QRS_NEXT_CUT()
PTP {E1 35817.24,E2 35817.24}
PTP {X 0,Y 759.922,A -85,B 0,C 180,E1 35817.24,E2 35817.24,E3 0,E4 0,E5 0,E6 0}
QRS_SPEED_INIT()
LIN {X 0,Y 759.922,Z 1164.5,A -85,B 0,C 180,E1 35817.24,E2 35817.24,E3 0,E4 0,E5 0,E6 0} C_VEL
LIN {X 0,Y 759.922,Z 407.653,A -85,B 0,C 180,E1 35817.24,E2 35817.24} C_VEL
LIN {X 0,Y 759.922,Z 399.576,A -85,B 0,C 180,E1 35817.24,E2 35817.24} C_VEL
LIN {X 0,Y 759.901,Z 397.576,A -85,B 0,C 180,E1 35817.09,E2 35817.09} C_VEL
LIN {X 0,Y 759.872,Z 397.569,A -85,B 0,C 180,E1 35814.336,E2 35814.336} C_VEL
LIN {X 0,Y 759.909,Z 397.568,A -85,B 0,C 180,E1 35811.602,E2 35811.602} C_VEL
LIN {X 0,Y 759.872,Z 397.574,A -85,B 0,C 180,E1 35808.77,E2 35808.77} C_VEL
LIN {X 0,Y 759.865,Z 397.569,A -85,B 0,C 180,E1 35806.143,E2 35806.143} C_VEL
LIN {X 0,Y 759.911,Z 397.573,A -85,B 0,C 180,E1 35803.317,E2 35803.317} C_VEL
LIN {X 0,Y 759.856,Z 397.573,A -85,B 0,C 180,E1 35800.554,E2 35800.554} C_VEL
LIN {X 0,Y 759.853,Z 397.571,A -85,B 0,C 180,E1 35798.055,E2 35798.055} C_VEL
LIN {X 0,Y 759.916,Z 397.57,A -85,B 0,C 180,E1 35795.348,E2 35795.348} C_VEL
LIN {X 0,Y 759.849,Z 397.574,A -85,B 0,C 180,E1 35792.489,E2 35792.489} C_VEL
LIN {X 0,Y 759.837,Z 397.573,A -85,B 0,C 180,E1 35790.083,E2 35790.083} C_VEL
LIN {X 0,Y 759.879,Z 397.571,A -85,B 0,C 180,E1 35787.508,E2 35787.508} C_VEL
LIN {X 0,Y 759.851,Z 397.576,A -85,B 0,C 180,E1 35784.527,E2 35784.527} C_VEL
LIN {X 0,Y 759.826,Z 397.575,A -85,B 0,C 180,E1 35782.146,E2 35782.146} C_VEL
LIN {X 0,Y 759.824,Z 397.574,A -85,B 0,C 180,E1 35779.848,E2 35779.848} C_VEL
LIN {X 0,Y 759.866,Z 397.572,A -85,B 0,C 180,E1 35777.337,E2 35777.337} C_VEL
LIN {X 0,Y 759.837,Z 397.577,A -85,B 0,C 180,E1 35774.393,E2 35774.393} C_VEL
LIN {X 0,Y 759.811,Z 397.575,A -85,B 0,C 180,E1 35772.054,E2 35772.054} C_VEL
LIN {X 0,Y 759.805,Z 397.577,A -85,B 0,C 180,E1 35769.777,E2 35769.777} C_VEL
LIN {X 0,Y 759.812,Z 397.577,A -85,B 0,C 180,E1 35767.539,E2 35767.539} C_VEL
LIN {X 0,Y 759.907,Z 397.578,A -85,B 0,C 180,E1 35764.808,E2 35764.808} C_VEL
LIN {X 0,Y 759.82,Z 397.573,A -85,B 0,C 180,E1 35762.061,E2 35762.061} C_VEL
LIN {X 0,Y 759.89,Z 397.819,A -85,B 0,C 180,E1 35760.915,E2 35760.915} C_VEL
LIN {X 0,Y 759.919,Z 413.781,A -85,B 0,C 180,E1 35759.761,E2 35759.761} C_VEL
LIN {X 0,Y 759.908,Z 637.992,A -85,B 0,C 180,E1 35757.315,E2 35757.315} C_VEL
LIN {X 0,Y 759.91,Z 802.101,A -85,B 0,C 180,E1 35755.549,E2 35755.549} C_VEL
LIN {X 0,Y 759.898,Z 825.96,A -85,B 0,C 180,E1 35755.172,E2 35755.172} C_VEL
LIN {X 0,Y 759.907,Z 847.797,A -85,B 0,C 180,E1 35754.694,E2 35754.694} C_VEL
LIN {X 0,Y 759.894,Z 868.493,A -85,B 0,C 180,E1 35754.136,E2 35754.136} C_VEL
LIN {X 0,Y 759.918,Z 893.54,A -85,B 0,C 180,E1 35753.303,E2 35753.303} C_VEL
LIN {X 0,Y 759.919,Z 913.093,A -85,B 0,C 180,E1 35752.529,E2 35752.529} C_VEL
LIN {X 0,Y 759.914,Z 935.14,A -85,B 0,C 180,E1 35751.523,E2 35751.523} C_VEL
LIN {X 0,Y 759.917,Z 955.453,A -85,B 0,C 180,E1 35750.439,E2 35750.439} C_VEL
LIN {X 0,Y 759.91,Z 975.283,A -85,B 0,C 180,E1 35749.245,E2 35749.245} C_VEL
LIN {X 0,Y 759.904,Z 994.198,A -85,B 0,C 180,E1 35747.933,E2 35747.933} C_VEL
LIN {X 0,Y 759.914,Z 1012.37,A -85,B 0,C 180,E1 35746.512,E2 35746.512} C_VEL
LIN {X 0,Y 759.91,Z 1028.199,A -85,B 0,C 180,E1 35745.102,E2 35745.102} C_VEL
LIN {X 0,Y 759.917,Z 1044.372,A -85,B 0,C 180,E1 35743.468,E2 35743.468} C_VEL
LIN {X 0,Y 759.904,Z 1057.076,A -85,B 0,C 180,E1 35741.999,E2 35741.999} C_VEL
LIN {X 0,Y 759.918,Z 1069.916,A -85,B 0,C 180,E1 35740.308,E2 35740.308} C_VEL
LIN {X 0,Y 759.893,Z 1080.292,A -85,B 0,C 180,E1 35738.704,E2 35738.704} C_VEL
LIN {X 0,Y 759.899,Z 1089.216,A -85,B 0,C 180,E1 35737.105,E2 35737.105} C_VEL
LIN {X 0,Y 759.897,Z 1097.567,A -85,B 0,C 180,E1 35735.285,E2 35735.285} C_VEL
LIN {X 0,Y 759.897,Z 1103.433,A -85,B 0,C 180,E1 35733.697,E2 35733.697} C_VEL
LIN {X 0,Y 759.914,Z 1108.651,A -85,B 0,C 180,E1 35731.885,E2 35731.885} C_VEL
LIN {X 0,Y 759.917,Z 1112.079,A -85,B 0,C 180,E1 35730.075,E2 35730.075} C_VEL
LIN {X 0,Y 759.889,Z 1113.939,A -85,B 0,C 180,E1 35728.417,E2 35728.417} C_VEL
LIN {X 0,Y 759.889,Z 1114.381,A -85,B 0,C 180,E1 35726.53,E2 35726.53} C_VEL
LIN {X 0,Y 759.892,Z 1113.442,A -85,B 0,C 180,E1 35724.932,E2 35724.932} C_VEL
LIN {X 0,Y 759.883,Z 1110.795,A -85,B 0,C 180,E1 35723.047,E2 35723.047} C_VEL
LIN {X 0,Y 759.909,Z 1106.908,A -85,B 0,C 180,E1 35721.373,E2 35721.373} C_VEL
LIN {X 0,Y 759.912,Z 1101.686,A -85,B 0,C 180,E1 35719.691,E2 35719.691} C_VEL
LIN {X 0,Y 759.905,Z 1094.199,A -85,B 0,C 180,E1 35717.847,E2 35717.847} C_VEL
LIN {X 0,Y 759.897,Z 1086.525,A -85,B 0,C 180,E1 35716.299,E2 35716.299} C_VEL
LIN {X 0,Y 759.904,Z 1076.531,A -85,B 0,C 180,E1 35714.586,E2 35714.586} C_VEL
LIN {X 0,Y 759.889,Z 1065.053,A -85,B 0,C 180,E1 35712.936,E2 35712.936} C_VEL
LIN {X 0,Y 759.913,Z 1052.308,A -85,B 0,C 180,E1 35711.33,E2 35711.33} C_VEL
LIN {X 0,Y 759.904,Z 1037.754,A -85,B 0,C 180,E1 35709.748,E2 35709.748} C_VEL
LIN {X 0,Y 759.9,Z 1021.891,A -85,B 0,C 180,E1 35708.219,E2 35708.219} C_VEL
LIN {X 0,Y 759.904,Z 1004.859,A -85,B 0,C 180,E1 35706.791,E2 35706.791} C_VEL
LIN {X 0,Y 759.918,Z 986.667,A -85,B 0,C 180,E1 35705.431,E2 35705.431} C_VEL
LIN {X 0,Y 759.913,Z 968.159,A -85,B 0,C 180,E1 35704.223,E2 35704.223} C_VEL
LIN {X 0,Y 759.916,Z 947.899,A -85,B 0,C 180,E1 35703.045,E2 35703.045} C_VEL
LIN {X 0,Y 759.916,Z 926.843,A -85,B 0,C 180,E1 35701.994,E2 35701.994} C_VEL
LIN {X 0,Y 759.917,Z 907.016,A -85,B 0,C 180,E1 35701.125,E2 35701.125} C_VEL
LIN {X 0,Y 759.905,Z 883.717,A -85,B 0,C 180,E1 35700.26,E2 35700.26} C_VEL
LIN {X 0,Y 759.899,Z 865.074,A -85,B 0,C 180,E1 35699.676,E2 35699.676} C_VEL
LIN {X 0,Y 759.905,Z 844.11,A -85,B 0,C 180,E1 35699.125,E2 35699.125} C_VEL
LIN {X 0,Y 759.903,Z 819.274,A -85,B 0,C 180,E1 35698.621,E2 35698.621} C_VEL
LIN {X 0,Y 759.908,Z 798.856,A -85,B 0,C 180,E1 35698.32,E2 35698.32} C_VEL
LIN {X 0,Y 759.909,Z 526.746,A -85,B 0,C 180,E1 35695.394,E2 35695.394} C_VEL
LIN {X 0,Y 759.919,Z 413.481,A -85,B 0,C 180,E1 35694.138,E2 35694.138} C_VEL
LIN {X 0,Y 759.888,Z 397.79,A -85,B 0,C 180,E1 35692.99,E2 35692.99} C_VEL
LIN {X 0,Y 759.814,Z 397.578,A -85,B 0,C 180,E1 35690.437,E2 35690.437} C_VEL
LIN {X 0,Y 759.804,Z 397.578,A -85,B 0,C 180,E1 35688.146,E2 35688.146} C_VEL
LIN {X 0,Y 759.81,Z 397.577,A -85,B 0,C 180,E1 35685.881,E2 35685.881} C_VEL
LIN {X 0,Y 759.854,Z 397.577,A -85,B 0,C 180,E1 35683.416,E2 35683.416} C_VEL
LIN {X 0,Y 759.844,Z 397.575,A -85,B 0,C 180,E1 35680.447,E2 35680.447} C_VEL
LIN {X 0,Y 759.824,Z 397.575,A -85,B 0,C 180,E1 35678.099,E2 35678.099} C_VEL
LIN {X 0,Y 759.824,Z 397.573,A -85,B 0,C 180,E1 35675.843,E2 35675.843} C_VEL
LIN {X 0,Y 759.857,Z 397.576,A -85,B 0,C 180,E1 35673.37,E2 35673.37} C_VEL
LIN {X 0,Y 759.862,Z 397.57,A -85,B 0,C 180,E1 35670.319,E2 35670.319} C_VEL
LIN {X 0,Y 759.836,Z 397.573,A -85,B 0,C 180,E1 35667.833,E2 35667.833} C_VEL
LIN {X 0,Y 759.853,Z 397.575,A -85,B 0,C 180,E1 35665.403,E2 35665.403} C_VEL
LIN {X 0,Y 759.919,Z 397.568,A -85,B 0,C 180,E1 35662.513,E2 35662.513} C_VEL
LIN {X 0,Y 759.85,Z 397.571,A -85,B 0,C 180,E1 35659.801,E2 35659.801} C_VEL
LIN {X 0,Y 759.87,Z 397.575,A -85,B 0,C 180,E1 35657.222,E2 35657.222} C_VEL
LIN {X 0,Y 759.906,Z 397.567,A -85,B 0,C 180,E1 35654.244,E2 35654.244} C_VEL
LIN {X 0,Y 759.858,Z 397.571,A -85,B 0,C 180,E1 35651.538,E2 35651.538} C_VEL
LIN {X 0,Y 759.917,Z 397.577,A -85,B 0,C 180,E1 35648.78,E2 35648.78} C_VEL
LIN {X 0,Y 759.881,Z 397.567,A -85,B 0,C 180,E1 35645.815,E2 35645.815} C_VEL
LIN {X 0,Y 759.887,Z 397.575,A -85,B 0,C 180,E1 35643.017,E2 35643.017} C_VEL
LIN {X 0,Y 759.92,Z 397.564,A -85,B 0,C 180,E1 35640,E2 35640} C_VEL
LIN {X 0,Y 759.876,Z 397.571,A -85,B 0,C 180,E1 35637.209,E2 35637.209} C_VEL
LIN {X 0,Y 759.905,Z 397.574,A -85,B 0,C 180,E1 35634.488,E2 35634.488} C_VEL
LIN {X 0,Y 759.896,Z 397.565,A -85,B 0,C 180,E1 35631.601,E2 35631.601} C_VEL
LIN {X 0,Y 759.911,Z 397.577,A -85,B 0,C 180,E1 35628.694,E2 35628.694} C_VEL
LIN {X 0,Y 759.918,Z 397.563,A -85,B 0,C 180,E1 35625.678,E2 35625.678} C_VEL
LIN {X 0,Y 759.914,Z 397.577,A -85,B 0,C 180,E1 35622.621,E2 35622.621} C_VEL
LIN {X 0,Y 759.911,Z 397.564,A -85,B 0,C 180,E1 35619.593,E2 35619.593} C_VEL
LIN {X 0,Y 759.914,Z 397.577,A -85,B 0,C 180,E1 35616.586,E2 35616.586} C_VEL
LIN {X 0,Y 759.895,Z 397.565,A -85,B 0,C 180,E1 35613.648,E2 35613.648} C_VEL
LIN {X 0,Y 759.902,Z 397.574,A -85,B 0,C 180,E1 35610.738,E2 35610.738} C_VEL
LIN {X 0,Y 759.877,Z 397.571,A -85,B 0,C 180,E1 35607.932,E2 35607.932} C_VEL
LIN {X 0,Y 759.912,Z 397.565,A -85,B 0,C 180,E1 35605.176,E2 35605.176} C_VEL
LIN {X 0,Y 759.896,Z 397.575,A -85,B 0,C 180,E1 35602.262,E2 35602.262} C_VEL
LIN {X 0,Y 759.879,Z 397.568,A -85,B 0,C 180,E1 35599.456,E2 35599.456} C_VEL
LIN {X 0,Y 759.91,Z 397.573,A -85,B 0,C 180,E1 35596.579,E2 35596.579} C_VEL
LIN {X 0,Y 759.863,Z 397.573,A -85,B 0,C 180,E1 35593.801,E2 35593.801} C_VEL
LIN {X 0,Y 759.896,Z 397.567,A -85,B 0,C 180,E1 35591.064,E2 35591.064} C_VEL
LIN {X 0,Y 759.886,Z 397.575,A -85,B 0,C 180,E1 35588.105,E2 35588.105} C_VEL
LIN {X 0,Y 759.913,Z 397.781,A -85,B 0,C 180,E1 35586.49,E2 35586.49} C_VEL
LIN {X 0,Y 759.908,Z 427.098,A -85,B 0,C 180,E1 35584.501,E2 35584.501} C_VEL
LIN {X 0,Y 759.907,Z 453.003,A -85,B 0,C 180,E1 35582.815,E2 35582.815} C_VEL
LIN {X 0,Y 759.893,Z 698.451,A -85,B 0,C 180,E1 35580.142,E2 35580.142} C_VEL
LIN {X 0,Y 759.92,Z 841.979,A -85,B 0,C 180,E1 35578.595,E2 35578.595} C_VEL
LIN {X 0,Y 759.894,Z 866.292,A -85,B 0,C 180,E1 35578.211,E2 35578.211} C_VEL
LIN {X 0,Y 759.9,Z 887.681,A -85,B 0,C 180,E1 35577.742,E2 35577.742} C_VEL
LIN {X 0,Y 759.897,Z 907.094,A -85,B 0,C 180,E1 35577.221,E2 35577.221} C_VEL
LIN {X 0,Y 759.919,Z 929.734,A -85,B 0,C 180,E1 35576.491,E2 35576.491} C_VEL
LIN {X 0,Y 759.916,Z 951.248,A -85,B 0,C 180,E1 35575.652,E2 35575.652} C_VEL
LIN {X 0,Y 759.913,Z 970.659,A -85,B 0,C 180,E1 35574.783,E2 35574.783} C_VEL
LIN {X 0,Y 759.91,Z 993.058,A -85,B 0,C 180,E1 35573.62,E2 35573.62} C_VEL
LIN {X 0,Y 759.92,Z 1011.704,A -85,B 0,C 180,E1 35572.513,E2 35572.513} C_VEL
LIN {X 0,Y 759.906,Z 1031.522,A -85,B 0,C 180,E1 35571.173,E2 35571.173} C_VEL
LIN {X 0,Y 759.916,Z 1048.884,A -85,B 0,C 180,E1 35569.845,E2 35569.845} C_VEL
LIN {X 0,Y 759.917,Z 1065.39,A -85,B 0,C 180,E1 35568.409,E2 35568.409} C_VEL
LIN {X 0,Y 759.895,Z 1079.946,A -85,B 0,C 180,E1 35566.985,E2 35566.985} C_VEL
LIN {X 0,Y 759.899,Z 1094.876,A -85,B 0,C 180,E1 35565.312,E2 35565.312} C_VEL
LIN {X 0,Y 759.905,Z 1106.572,A -85,B 0,C 180,E1 35563.815,E2 35563.815} C_VEL
LIN {X 0,Y 759.9,Z 1118.785,A -85,B 0,C 180,E1 35561.999,E2 35561.999} C_VEL
LIN {X 0,Y 759.907,Z 1127.555,A -85,B 0,C 180,E1 35560.462,E2 35560.462} C_VEL
LIN {X 0,Y 759.888,Z 1136.073,A -85,B 0,C 180,E1 35558.704,E2 35558.704} C_VEL
LIN {X 0,Y 759.918,Z 1142.726,A -85,B 0,C 180,E1 35556.953,E2 35556.953} C_VEL
LIN {X 0,Y 759.883,Z 1147.51,A -85,B 0,C 180,E1 35555.361,E2 35555.361} C_VEL
LIN {X 0,Y 759.919,Z 1151.559,A -85,B 0,C 180,E1 35553.47,E2 35553.47} C_VEL
LIN {X 0,Y 759.902,Z 1153.63,A -85,B 0,C 180,E1 35551.81,E2 35551.81} C_VEL
LIN {X 0,Y 759.92,Z 1154.5,A -85,B 0,C 180,E1 35550,E2 35550} C_VEL
LIN {X 0,Y 759.902,Z 1153.63,A -85,B 0,C 180,E1 35548.19,E2 35548.19} C_VEL
LIN {X 0,Y 759.919,Z 1151.559,A -85,B 0,C 180,E1 35546.53,E2 35546.53} C_VEL
LIN {X 0,Y 759.883,Z 1147.51,A -85,B 0,C 180,E1 35544.639,E2 35544.639} C_VEL
LIN {X 0,Y 759.918,Z 1142.726,A -85,B 0,C 180,E1 35543.047,E2 35543.047} C_VEL
LIN {X 0,Y 759.889,Z 1135.729,A -85,B 0,C 180,E1 35541.22,E2 35541.22} C_VEL
LIN {X 0,Y 759.907,Z 1127.555,A -85,B 0,C 180,E1 35539.538,E2 35539.538} C_VEL
LIN {X 0,Y 759.9,Z 1118.785,A -85,B 0,C 180,E1 35538.001,E2 35538.001} C_VEL
LIN {X 0,Y 759.904,Z 1106.265,A -85,B 0,C 180,E1 35536.144,E2 35536.144} C_VEL
LIN {X 0,Y 759.9,Z 1094.679,A -85,B 0,C 180,E1 35534.664,E2 35534.664} C_VEL
LIN {X 0,Y 759.896,Z 1079.169,A -85,B 0,C 180,E1 35532.937,E2 35532.937} C_VEL
LIN {X 0,Y 759.914,Z 1064.539,A -85,B 0,C 180,E1 35531.512,E2 35531.512} C_VEL
LIN {X 0,Y 759.913,Z 1046.484,A -85,B 0,C 180,E1 35529.965,E2 35529.965} C_VEL
LIN {X 0,Y 759.91,Z 1029.578,A -85,B 0,C 180,E1 35528.684,E2 35528.684} C_VEL
LIN {X 0,Y 759.918,Z 1009.719,A -85,B 0,C 180,E1 35527.364,E2 35527.364} C_VEL
LIN {X 0,Y 759.91,Z 990.877,A -85,B 0,C 180,E1 35526.257,E2 35526.257} C_VEL
LIN {X 0,Y 759.913,Z 969.006,A -85,B 0,C 180,E1 35525.14,E2 35525.14} C_VEL
LIN {X 0,Y 759.917,Z 950.063,A -85,B 0,C 180,E1 35524.299,E2 35524.299} C_VEL
LIN {X 0,Y 759.915,Z 927.316,A -85,B 0,C 180,E1 35523.425,E2 35523.425} C_VEL
LIN {X 0,Y 759.899,Z 906.002,A -85,B 0,C 180,E1 35522.748,E2 35522.748} C_VEL
LIN {X 0,Y 759.898,Z 886.063,A -85,B 0,C 180,E1 35522.218,E2 35522.218} C_VEL
LIN {X 0,Y 759.898,Z 861.401,A -85,B 0,C 180,E1 35521.701,E2 35521.701} C_VEL
LIN {X 0,Y 759.92,Z 840.267,A -85,B 0,C 180,E1 35521.383,E2 35521.383} C_VEL
LIN {X 0,Y 759.85,Z 582.634,A -85,B 0,C 180,E1 35518.608,E2 35518.608} C_VEL
LIN {X 0,Y 759.905,Z 452.847,A -85,B 0,C 180,E1 35517.179,E2 35517.179} C_VEL
LIN {X 0,Y 759.916,Z 411.18,A -85,B 0,C 180,E1 35514.438,E2 35514.438} C_VEL
LIN {X 0,Y 759.913,Z 397.769,A -85,B 0,C 180,E1 35513.506,E2 35513.506} C_VEL
LIN {X 0,Y 759.864,Z 397.57,A -85,B 0,C 180,E1 35510.691,E2 35510.691} C_VEL
LIN {X 0,Y 759.871,Z 397.575,A -85,B 0,C 180,E1 35508.028,E2 35508.028} C_VEL
LIN {X 0,Y 759.912,Z 397.568,A -85,B 0,C 180,E1 35505.149,E2 35505.149} C_VEL
LIN {X 0,Y 759.866,Z 397.57,A -85,B 0,C 180,E1 35502.356,E2 35502.356} C_VEL
LIN {X 0,Y 759.915,Z 397.578,A -85,B 0,C 180,E1 35499.551,E2 35499.551} C_VEL
LIN {X 0,Y 759.892,Z 397.566,A -85,B 0,C 180,E1 35496.589,E2 35496.589} C_VEL
LIN {X 0,Y 759.894,Z 397.575,A -85,B 0,C 180,E1 35493.73,E2 35493.73} C_VEL
LIN {X 0,Y 759.909,Z 397.565,A -85,B 0,C 180,E1 35490.771,E2 35490.771} C_VEL
LIN {X 0,Y 759.881,Z 397.57,A -85,B 0,C 180,E1 35488.001,E2 35488.001} C_VEL
LIN {X 0,Y 759.902,Z 397.573,A -85,B 0,C 180,E1 35485.235,E2 35485.235} C_VEL
LIN {X 0,Y 759.9,Z 397.565,A -85,B 0,C 180,E1 35482.328,E2 35482.328} C_VEL
LIN {X 0,Y 759.911,Z 397.577,A -85,B 0,C 180,E1 35479.364,E2 35479.364} C_VEL
LIN {X 0,Y 759.915,Z 397.563,A -85,B 0,C 180,E1 35476.355,E2 35476.355} C_VEL
LIN {X 0,Y 759.915,Z 397.577,A -85,B 0,C 180,E1 35473.313,E2 35473.313} C_VEL
LIN {X 0,Y 759.91,Z 397.564,A -85,B 0,C 180,E1 35470.309,E2 35470.309} C_VEL
LIN {X 0,Y 759.913,Z 397.577,A -85,B 0,C 180,E1 35467.257,E2 35467.257} C_VEL
LIN {X 0,Y 759.89,Z 397.566,A -85,B 0,C 180,E1 35464.377,E2 35464.377} C_VEL
LIN {X 0,Y 759.904,Z 397.573,A -85,B 0,C 180,E1 35461.508,E2 35461.508} C_VEL
LIN {X 0,Y 759.876,Z 397.572,A -85,B 0,C 180,E1 35458.794,E2 35458.794} C_VEL
LIN {X 0,Y 759.901,Z 397.576,A -85,B 0,C 180,E1 35457.09,E2 35457.09} C_VEL
LIN {X 0,Y 758.866,Z 397.696,A -85,B 0,C 180,E1 35456.509,E2 35456.509} C_VEL
LIN {X 0,Y 752.45,Z 398.503,A -85,B 0,C 180,E1 35454.882,E2 35454.882} C_VEL
LIN {X 0,Y 751.929,Z 398.559,A -85,B 0,C 180,E1 35454.46,E2 35454.46} C_VEL
LIN {X 0,Y 751.974,Z 398.554,A -85,B 0,C 180,E1 35451.743,E2 35451.743} C_VEL
LIN {X 0,Y 751.937,Z 398.563,A -85,B 0,C 180,E1 35448.805,E2 35448.805} C_VEL
LIN {X 0,Y 751.929,Z 398.557,A -85,B 0,C 180,E1 35446.105,E2 35446.105} C_VEL
LIN {X 0,Y 751.975,Z 398.564,A -85,B 0,C 180,E1 35443.212,E2 35443.212} C_VEL
LIN {X 0,Y 751.915,Z 398.562,A -85,B 0,C 180,E1 35440.502,E2 35440.502} C_VEL
LIN {X 0,Y 751.922,Z 398.559,A -85,B 0,C 180,E1 35437.951,E2 35437.951} C_VEL
LIN {X 0,Y 751.977,Z 398.564,A -85,B 0,C 180,E1 35435.07,E2 35435.07} C_VEL
LIN {X 0,Y 751.903,Z 398.562,A -85,B 0,C 180,E1 35432.333,E2 35432.333} C_VEL
LIN {X 0,Y 751.905,Z 398.561,A -85,B 0,C 180,E1 35429.911,E2 35429.911} C_VEL
LIN {X 0,Y 751.979,Z 398.562,A -85,B 0,C 180,E1 35427.145,E2 35427.145} C_VEL
LIN {X 0,Y 751.897,Z 398.564,A -85,B 0,C 180,E1 35424.344,E2 35424.344} C_VEL
LIN {X 0,Y 751.886,Z 398.564,A -85,B 0,C 180,E1 35421.996,E2 35421.996} C_VEL
LIN {X 0,Y 751.899,Z 398.563,A -85,B 0,C 180,E1 35419.637,E2 35419.637} C_VEL
LIN {X 0,Y 751.953,Z 398.566,A -85,B 0,C 180,E1 35416.777,E2 35416.777} C_VEL
LIN {X 0,Y 751.881,Z 398.566,A -85,B 0,C 180,E1 35414.175,E2 35414.175} C_VEL
LIN {X 0,Y 751.87,Z 398.561,A -85,B 0,C 180,E1 35411.864,E2 35411.864} C_VEL
LIN {X 0,Y 751.878,Z 398.567,A -85,B 0,C 180,E1 35409.527,E2 35409.527} C_VEL
LIN {X 0,Y 751.953,Z 398.568,A -85,B 0,C 180,E1 35406.695,E2 35406.695} C_VEL
LIN {X 0,Y 751.876,Z 398.568,A -85,B 0,C 180,E1 35404.047,E2 35404.047} C_VEL
LIN {X 0,Y 751.871,Z 398.558,A -85,B 0,C 180,E1 35401.811,E2 35401.811} C_VEL
LIN {X 0,Y 751.955,Z 398.922,A -85,B 0,C 180,E1 35401.234,E2 35401.234} C_VEL
LIN {X 0,Y 752.71,Z 402.275,A -85,B 0,C 180,E1 35400.937,E2 35400.937} C_VEL
LIN {X 0,Y 752.755,Z 413.762,A -85,B 0,C 180,E1 35400.114,E2 35400.114} C_VEL
LIN {X 0,Y 753.183,Z 417.042,A -85,B 0,C 180,E1 35400.046,E2 35400.046} C_VEL
LIN {X 0,Y 752.967,Z 667.075,A -85,B 0,C 180,E1 35397.31,E2 35397.31} C_VEL
LIN {X 0,Y 752.873,Z 802.384,A -85,B 0,C 180,E1 35395.838,E2 35395.838} C_VEL
LIN {X 0,Y 752.802,Z 827.22,A -85,B 0,C 180,E1 35395.436,E2 35395.436} C_VEL
LIN {X 0,Y 752.759,Z 848.615,A -85,B 0,C 180,E1 35394.96,E2 35394.96} C_VEL
LIN {X 0,Y 752.686,Z 870.446,A -85,B 0,C 180,E1 35394.361,E2 35394.361} C_VEL
LIN {X 0,Y 752.612,Z 894.301,A -85,B 0,C 180,E1 35393.55,E2 35393.55} C_VEL
LIN {X 0,Y 752.545,Z 914.316,A -85,B 0,C 180,E1 35392.746,E2 35392.746} C_VEL
LIN {X 0,Y 752.433,Z 937.119,A -85,B 0,C 180,E1 35391.68,E2 35391.68} C_VEL
LIN {X 0,Y 752.364,Z 955.766,A -85,B 0,C 180,E1 35390.671,E2 35390.671} C_VEL
LIN {X 0,Y 752.265,Z 976.401,A -85,B 0,C 180,E1 35389.408,E2 35389.408} C_VEL
LIN {X 0,Y 752.195,Z 994.827,A -85,B 0,C 180,E1 35388.112,E2 35388.112} C_VEL
LIN {X 0,Y 752.126,Z 1013.684,A -85,B 0,C 180,E1 35386.608,E2 35386.608} C_VEL
LIN {X 0,Y 752.076,Z 1029.403,A -85,B 0,C 180,E1 35385.184,E2 35385.184} C_VEL
LIN {X 0,Y 752.026,Z 1045.376,A -85,B 0,C 180,E1 35383.533,E2 35383.533} C_VEL
LIN {X 0,Y 751.983,Z 1057.987,A -85,B 0,C 180,E1 35382.05,E2 35382.05} C_VEL
LIN {X 0,Y 751.962,Z 1071.168,A -85,B 0,C 180,E1 35380.264,E2 35380.264} C_VEL
LIN {X 0,Y 751.923,Z 1080.95,A -85,B 0,C 180,E1 35378.719,E2 35378.719} C_VEL
LIN {X 0,Y 751.904,Z 1090.572,A -85,B 0,C 180,E1 35376.951,E2 35376.951} C_VEL
LIN {X 0,Y 751.912,Z 1098.3,A -85,B 0,C 180,E1 35375.188,E2 35375.188} C_VEL
LIN {X 0,Y 751.892,Z 1104.048,A -85,B 0,C 180,E1 35373.583,E2 35373.583} C_VEL
LIN {X 0,Y 751.914,Z 1109.351,A -85,B 0,C 180,E1 35371.6,E2 35371.6} C_VEL
LIN {X 0,Y 751.914,Z 1112.352,A -85,B 0,C 180,E1 35369.924,E2 35369.924} C_VEL
LIN {X 0,Y 751.917,Z 1114.196,A -85,B 0,C 180,E1 35368.019,E2 35368.019} C_VEL
LIN {X 0,Y 751.889,Z 1114.327,A -85,B 0,C 180,E1 35366.34,E2 35366.34} C_VEL
LIN {X 0,Y 751.911,Z 1113.154,A -85,B 0,C 180,E1 35364.582,E2 35364.582} C_VEL
LIN {X 0,Y 751.884,Z 1110.249,A -85,B 0,C 180,E1 35362.742,E2 35362.742} C_VEL
LIN {X 0,Y 751.916,Z 1106.613,A -85,B 0,C 180,E1 35361.203,E2 35361.203} C_VEL
LIN {X 0,Y 751.902,Z 1100.739,A -85,B 0,C 180,E1 35359.339,E2 35359.339} C_VEL
LIN {X 0,Y 751.915,Z 1093.328,A -85,B 0,C 180,E1 35357.559,E2 35357.559} C_VEL
LIN {X 0,Y 751.921,Z 1085.11,A -85,B 0,C 180,E1 35355.916,E2 35355.916} C_VEL
LIN {X 0,Y 751.944,Z 1074.199,A -85,B 0,C 180,E1 35354.102,E2 35354.102} C_VEL
LIN {X 0,Y 751.96,Z 1063.623,A -85,B 0,C 180,E1 35352.591,E2 35352.591} C_VEL
LIN {X 0,Y 751.998,Z 1049.393,A -85,B 0,C 180,E1 35350.827,E2 35350.827} C_VEL
LIN {X 0,Y 752.048,Z 1035.881,A -85,B 0,C 180,E1 35349.37,E2 35349.37} C_VEL
LIN {X 0,Y 752.119,Z 1019.142,A -85,B 0,C 180,E1 35347.776,E2 35347.776} C_VEL
LIN {X 0,Y 752.158,Z 1002.853,A -85,B 0,C 180,E1 35346.413,E2 35346.413} C_VEL
LIN {X 0,Y 752.247,Z 983.216,A -85,B 0,C 180,E1 35344.966,E2 35344.966} C_VEL
LIN {X 0,Y 752.312,Z 965.042,A -85,B 0,C 180,E1 35343.785,E2 35343.785} C_VEL
LIN {X 0,Y 752.417,Z 943.077,A -85,B 0,C 180,E1 35342.54,E2 35342.54} C_VEL
LIN {X 0,Y 752.49,Z 923.974,A -85,B 0,C 180,E1 35341.595,E2 35341.595} C_VEL
LIN {X 0,Y 752.6,Z 900.73,A -85,B 0,C 180,E1 35340.604,E2 35340.604} C_VEL
LIN {X 0,Y 752.644,Z 879.969,A -85,B 0,C 180,E1 35339.856,E2 35339.856} C_VEL
LIN {X 0,Y 752.741,Z 857.575,A -85,B 0,C 180,E1 35339.176,E2 35339.176} C_VEL
LIN {X 0,Y 752.792,Z 834.253,A -85,B 0,C 180,E1 35338.62,E2 35338.62} C_VEL
LIN {X 0,Y 752.846,Z 814.363,A -85,B 0,C 180,E1 35338.249,E2 35338.249} C_VEL
LIN {X 0,Y 752.88,Z 789.412,A -85,B 0,C 180,E1 35337.912,E2 35337.912} C_VEL
LIN {X 0,Y 753.078,Z 533.824,A -85,B 0,C 180,E1 35335.152,E2 35335.152} C_VEL
LIN {X 0,Y 752.996,Z 414.882,A -85,B 0,C 180,E1 35333.83,E2 35333.83} C_VEL
LIN {X 0,Y 752.683,Z 412.464,A -85,B 0,C 180,E1 35333.718,E2 35333.718} C_VEL
LIN {X 0,Y 752.569,Z 400.863,A -85,B 0,C 180,E1 35332.862,E2 35332.862} C_VEL
LIN {X 0,Y 751.903,Z 398.647,A -85,B 0,C 180,E1 35332.623,E2 35332.623} C_VEL
LIN {X 0,Y 751.87,Z 398.569,A -85,B 0,C 180,E1 35330.332,E2 35330.332} C_VEL
LIN {X 0,Y 751.866,Z 398.568,A -85,B 0,C 180,E1 35328.015,E2 35328.015} C_VEL
LIN {X 0,Y 751.89,Z 398.567,A -85,B 0,C 180,E1 35325.613,E2 35325.613} C_VEL
LIN {X 0,Y 751.926,Z 398.561,A -85,B 0,C 180,E1 35322.662,E2 35322.662} C_VEL
LIN {X 0,Y 751.884,Z 398.564,A -85,B 0,C 180,E1 35320.164,E2 35320.164} C_VEL
LIN {X 0,Y 751.883,Z 398.564,A -85,B 0,C 180,E1 35317.908,E2 35317.908} C_VEL
LIN {X 0,Y 751.902,Z 398.56,A -85,B 0,C 180,E1 35315.526,E2 35315.526} C_VEL
LIN {X 0,Y 751.966,Z 398.56,A -85,B 0,C 180,E1 35312.674,E2 35312.674} C_VEL
LIN {X 0,Y 751.899,Z 398.558,A -85,B 0,C 180,E1 35310.001,E2 35310.001} C_VEL
LIN {X 0,Y 751.903,Z 398.562,A -85,B 0,C 180,E1 35307.566,E2 35307.566} C_VEL
LIN {X 0,Y 751.977,Z 398.561,A -85,B 0,C 180,E1 35304.745,E2 35304.745} C_VEL
LIN {X 0,Y 751.912,Z 398.561,A -85,B 0,C 180,E1 35301.942,E2 35301.942} C_VEL
LIN {X 0,Y 751.916,Z 398.562,A -85,B 0,C 180,E1 35299.418,E2 35299.418} C_VEL
LIN {X 0,Y 751.974,Z 398.56,A -85,B 0,C 180,E1 35296.612,E2 35296.612} C_VEL
LIN {X 0,Y 751.926,Z 398.559,A -85,B 0,C 180,E1 35293.849,E2 35293.849} C_VEL
LIN {X 0,Y 751.933,Z 398.562,A -85,B 0,C 180,E1 35291.195,E2 35291.195} C_VEL
LIN {X 0,Y 751.974,Z 398.555,A -85,B 0,C 180,E1 35288.257,E2 35288.257} C_VEL
LIN {X 0,Y 751.927,Z 398.559,A -85,B 0,C 180,E1 35285.494,E2 35285.494} C_VEL
LIN {X 0,Y 751.973,Z 398.565,A -85,B 0,C 180,E1 35282.744,E2 35282.744} C_VEL
LIN {X 0,Y 751.953,Z 398.555,A -85,B 0,C 180,E1 35279.771,E2 35279.771} C_VEL
LIN {X 0,Y 751.959,Z 398.563,A -85,B 0,C 180,E1 35276.875,E2 35276.875} C_VEL
LIN {X 0,Y 751.972,Z 398.553,A -85,B 0,C 180,E1 35273.817,E2 35273.817} C_VEL
LIN {X 0,Y 751.956,Z 398.563,A -85,B 0,C 180,E1 35270.895,E2 35270.895} C_VEL
LIN {X 0,Y 751.96,Z 398.555,A -85,B 0,C 180,E1 35268.028,E2 35268.028} C_VEL
LIN {X 0,Y 751.95,Z 398.557,A -85,B 0,C 180,E1 35265.287,E2 35265.287} C_VEL
LIN {X 0,Y 751.965,Z 398.564,A -85,B 0,C 180,E1 35262.432,E2 35262.432} C_VEL
LIN {X 0,Y 751.97,Z 398.553,A -85,B 0,C 180,E1 35259.449,E2 35259.449} C_VEL
LIN {X 0,Y 751.97,Z 398.566,A -85,B 0,C 180,E1 35256.49,E2 35256.49} C_VEL
LIN {X 0,Y 751.97,Z 398.552,A -85,B 0,C 180,E1 35253.494,E2 35253.494} C_VEL
LIN {X 0,Y 751.969,Z 398.565,A -85,B 0,C 180,E1 35250.415,E2 35250.415} C_VEL
LIN {X 0,Y 751.958,Z 398.555,A -85,B 0,C 180,E1 35247.463,E2 35247.463} C_VEL
LIN {X 0,Y 751.977,Z 398.565,A -85,B 0,C 180,E1 35244.466,E2 35244.466} C_VEL
LIN {X 0,Y 751.933,Z 398.558,A -85,B 0,C 180,E1 35241.68,E2 35241.68} C_VEL
LIN {X 0,Y 751.972,Z 398.557,A -85,B 0,C 180,E1 35238.933,E2 35238.933} C_VEL
LIN {X 0,Y 751.936,Z 398.563,A -85,B 0,C 180,E1 35236.005,E2 35236.005} C_VEL
LIN {X 0,Y 751.936,Z 398.559,A -85,B 0,C 180,E1 35233.327,E2 35233.327} C_VEL
LIN {X 0,Y 751.98,Z 398.564,A -85,B 0,C 180,E1 35230.358,E2 35230.358} C_VEL
LIN {X 0,Y 751.915,Z 398.558,A -85,B 0,C 180,E1 35227.617,E2 35227.617} C_VEL
LIN {X 0,Y 752.001,Z 398.76,A -85,B 0,C 180,E1 35226.87,E2 35226.87} C_VEL
LIN {X 0,Y 752.898,Z 401.513,A -85,B 0,C 180,E1 35226.605,E2 35226.605} C_VEL
LIN {X 0,Y 752.709,Z 437.421,A -85,B 0,C 180,E1 35224.188,E2 35224.188} C_VEL
LIN {X 0,Y 752.768,Z 453.102,A -85,B 0,C 180,E1 35223.163,E2 35223.163} C_VEL
LIN {X 0,Y 753.18,Z 456.661,A -85,B 0,C 180,E1 35223.095,E2 35223.095} C_VEL
LIN {X 0,Y 752.958,Z 709.953,A -85,B 0,C 180,E1 35220.324,E2 35220.324} C_VEL
LIN {X 0,Y 752.883,Z 842.408,A -85,B 0,C 180,E1 35218.882,E2 35218.882} C_VEL
LIN {X 0,Y 752.798,Z 867.202,A -85,B 0,C 180,E1 35218.482,E2 35218.482} C_VEL
LIN {X 0,Y 752.752,Z 888.593,A -85,B 0,C 180,E1 35218.006,E2 35218.006} C_VEL
LIN {X 0,Y 752.69,Z 909.676,A -85,B 0,C 180,E1 35217.428,E2 35217.428} C_VEL
LIN {X 0,Y 752.612,Z 934.071,A -85,B 0,C 180,E1 35216.604,E2 35216.604} C_VEL
LIN {X 0,Y 752.542,Z 953.239,A -85,B 0,C 180,E1 35215.837,E2 35215.837} C_VEL
LIN {X 0,Y 752.445,Z 975.244,A -85,B 0,C 180,E1 35214.822,E2 35214.822} C_VEL
LIN {X 0,Y 752.361,Z 995.242,A -85,B 0,C 180,E1 35213.746,E2 35213.746} C_VEL
LIN {X 0,Y 752.282,Z 1015.599,A -85,B 0,C 180,E1 35212.507,E2 35212.507} C_VEL
LIN {X 0,Y 752.195,Z 1034.285,A -85,B 0,C 180,E1 35211.197,E2 35211.197} C_VEL
LIN {X 0,Y 752.117,Z 1052.744,A -85,B 0,C 180,E1 35209.735,E2 35209.735} C_VEL
LIN {X 0,Y 752.079,Z 1068.793,A -85,B 0,C 180,E1 35208.286,E2 35208.286} C_VEL
LIN {X 0,Y 752.023,Z 1085.09,A -85,B 0,C 180,E1 35206.611,E2 35206.611} C_VEL
LIN {X 0,Y 751.972,Z 1097.889,A -85,B 0,C 180,E1 35205.107,E2 35205.107} C_VEL
LIN {X 0,Y 751.94,Z 1111.231,A -85,B 0,C 180,E1 35203.3,E2 35203.3} C_VEL
LIN {X 0,Y 751.929,Z 1120.637,A -85,B 0,C 180,E1 35201.817,E2 35201.817} C_VEL
LIN {X 0,Y 751.917,Z 1130.399,A -85,B 0,C 180,E1 35200.032,E2 35200.032} C_VEL
LIN {X 0,Y 751.918,Z 1138.205,A -85,B 0,C 180,E1 35198.257,E2 35198.257} C_VEL
LIN {X 0,Y 751.904,Z 1144.144,A -85,B 0,C 180,E1 35196.599,E2 35196.599} C_VEL
LIN {X 0,Y 751.915,Z 1149.336,A -85,B 0,C 180,E1 35194.653,E2 35194.653} C_VEL
LIN {X 0,Y 751.883,Z 1152.234,A -85,B 0,C 180,E1 35193.049,E2 35193.049} C_VEL
LIN {X 0,Y 751.913,Z 1154.149,A -85,B 0,C 180,E1 35191.219,E2 35191.219} C_VEL
LIN {X 0,Y 751.881,Z 1154.351,A -85,B 0,C 180,E1 35189.467,E2 35189.467} C_VEL
LIN {X 0,Y 751.919,Z 1153.296,A -85,B 0,C 180,E1 35187.79,E2 35187.79} C_VEL
LIN {X 0,Y 751.915,Z 1150.287,A -85,B 0,C 180,E1 35185.806,E2 35185.806} C_VEL
LIN {X 0,Y 751.918,Z 1146.481,A -85,B 0,C 180,E1 35184.2,E2 35184.2} C_VEL
LIN {X 0,Y 751.888,Z 1140.637,A -85,B 0,C 180,E1 35182.358,E2 35182.358} C_VEL
LIN {X 0,Y 751.921,Z 1133.519,A -85,B 0,C 180,E1 35180.646,E2 35180.646} C_VEL
LIN {X 0,Y 751.905,Z 1125.516,A -85,B 0,C 180,E1 35179.038,E2 35179.038} C_VEL
LIN {X 0,Y 751.937,Z 1114.349,A -85,B 0,C 180,E1 35177.169,E2 35177.169} C_VEL
LIN {X 0,Y 751.977,Z 1103.95,A -85,B 0,C 180,E1 35175.681,E2 35175.681} C_VEL
LIN {X 0,Y 752.003,Z 1090.042,A -85,B 0,C 180,E1 35173.945,E2 35173.945} C_VEL
LIN {X 0,Y 752.049,Z 1076.064,A -85,B 0,C 180,E1 35172.434,E2 35172.434} C_VEL
LIN {X 0,Y 752.114,Z 1059.246,A -85,B 0,C 180,E1 35170.83,E2 35170.83} C_VEL
LIN {X 0,Y 752.168,Z 1042.806,A -85,B 0,C 180,E1 35169.455,E2 35169.455} C_VEL
LIN {X 0,Y 752.246,Z 1022.85,A -85,B 0,C 180,E1 35167.986,E2 35167.986} C_VEL
LIN {X 0,Y 752.314,Z 1004.43,A -85,B 0,C 180,E1 35166.792,E2 35166.792} C_VEL
LIN {X 0,Y 752.417,Z 983.14,A -85,B 0,C 180,E1 35165.588,E2 35165.588} C_VEL
LIN {X 0,Y 752.491,Z 963.796,A -85,B 0,C 180,E1 35164.632,E2 35164.632} C_VEL
LIN {X 0,Y 752.602,Z 939.818,A -85,B 0,C 180,E1 35163.614,E2 35163.614} C_VEL
LIN {X 0,Y 752.648,Z 919.683,A -85,B 0,C 180,E1 35162.892,E2 35162.892} C_VEL
LIN {X 0,Y 752.748,Z 897.171,A -85,B 0,C 180,E1 35162.209,E2 35162.209} C_VEL
LIN {X 0,Y 752.785,Z 874.082,A -85,B 0,C 180,E1 35161.661,E2 35161.661} C_VEL
LIN {X 0,Y 752.845,Z 854.281,A -85,B 0,C 180,E1 35161.293,E2 35161.293} C_VEL
LIN {X 0,Y 752.889,Z 829.297,A -85,B 0,C 180,E1 35160.956,E2 35160.956} C_VEL
LIN {X 0,Y 753.015,Z 587.065,A -85,B 0,C 180,E1 35158.339,E2 35158.339} C_VEL
LIN {X 0,Y 753.012,Z 454.234,A -85,B 0,C 180,E1 35156.869,E2 35156.869} C_VEL
LIN {X 0,Y 752.698,Z 451.927,A -85,B 0,C 180,E1 35156.772,E2 35156.772} C_VEL
LIN {X 0,Y 752.871,Z 412.01,A -85,B 0,C 180,E1 35154.11,E2 35154.11} C_VEL
LIN {X 0,Y 752.719,Z 401.07,A -85,B 0,C 180,E1 35153.354,E2 35153.354} C_VEL
LIN {X 0,Y 751.982,Z 398.663,A -85,B 0,C 180,E1 35153.105,E2 35153.105} C_VEL
LIN {X 0,Y 751.916,Z 398.563,A -85,B 0,C 180,E1 35150.335,E2 35150.335} C_VEL
LIN {X 0,Y 751.973,Z 398.566,A -85,B 0,C 180,E1 35147.56,E2 35147.56} C_VEL
LIN {X 0,Y 751.939,Z 398.558,A -85,B 0,C 180,E1 35144.649,E2 35144.649} C_VEL
LIN {X 0,Y 751.945,Z 398.562,A -85,B 0,C 180,E1 35141.87,E2 35141.87} C_VEL
LIN {X 0,Y 751.979,Z 398.554,A -85,B 0,C 180,E1 35138.874,E2 35138.874} C_VEL
LIN {X 0,Y 751.935,Z 398.56,A -85,B 0,C 180,E1 35136.051,E2 35136.051} C_VEL
LIN {X 0,Y 751.968,Z 398.562,A -85,B 0,C 180,E1 35133.31,E2 35133.31} C_VEL
LIN {X 0,Y 751.954,Z 398.556,A -85,B 0,C 180,E1 35130.439,E2 35130.439} C_VEL
LIN {X 0,Y 751.97,Z 398.565,A -85,B 0,C 180,E1 35127.512,E2 35127.512} C_VEL
LIN {X 0,Y 751.975,Z 398.551,A -85,B 0,C 180,E1 35124.511,E2 35124.511} C_VEL
LIN {X 0,Y 751.969,Z 398.565,A -85,B 0,C 180,E1 35121.531,E2 35121.531} C_VEL
LIN {X 0,Y 751.969,Z 398.553,A -85,B 0,C 180,E1 35118.53,E2 35118.53} C_VEL
LIN {X 0,Y 751.962,Z 398.563,A -85,B 0,C 180,E1 35115.581,E2 35115.581} C_VEL
LIN {X 0,Y 751.948,Z 398.558,A -85,B 0,C 180,E1 35112.752,E2 35112.752} C_VEL
LIN {X 0,Y 751.961,Z 398.556,A -85,B 0,C 180,E1 35109.954,E2 35109.954} C_VEL
LIN {X 0,Y 751.958,Z 398.564,A -85,B 0,C 180,E1 35107.104,E2 35107.104} C_VEL
LIN {X 0,Y 751.968,Z 398.553,A -85,B 0,C 180,E1 35104.194,E2 35104.194} C_VEL
LIN {X 0,Y 751.966,Z 398.565,A -85,B 0,C 180,E1 35101.143,E2 35101.143} C_VEL
LIN {X 0,Y 751.942,Z 398.556,A -85,B 0,C 180,E1 35098.324,E2 35098.324} C_VEL
LIN {X 0,Y 751.968,Z 398.56,A -85,B 0,C 180,E1 35095.5,E2 35095.5} C_VEL
LIN {X 0,Y 751.929,Z 398.559,A -85,B 0,C 180,E1 35094.46,E2 35094.46} C_VEL
LIN {X 0,Y 750.952,Z 398.684,A -85,B 0,C 180,E1 35093.873,E2 35093.873} C_VEL
LIN {X 0,Y 744.556,Z 399.477,A -85,B 0,C 180,E1 35092.229,E2 35092.229} C_VEL
LIN {X 0,Y 744.033,Z 399.542,A -85,B 0,C 180,E1 35091.802,E2 35091.802} C_VEL
LIN {X 0,Y 744,Z 399.552,A -85,B 0,C 180,E1 35088.837,E2 35088.837} C_VEL
LIN {X 0,Y 743.986,Z 399.545,A -85,B 0,C 180,E1 35086.159,E2 35086.159} C_VEL
LIN {X 0,Y 744.034,Z 399.552,A -85,B 0,C 180,E1 35083.286,E2 35083.286} C_VEL
LIN {X 0,Y 743.978,Z 399.551,A -85,B 0,C 180,E1 35080.53,E2 35080.53} C_VEL
LIN {X 0,Y 743.981,Z 399.549,A -85,B 0,C 180,E1 35077.978,E2 35077.978} C_VEL
LIN {X 0,Y 744.038,Z 399.551,A -85,B 0,C 180,E1 35075.11,E2 35075.11} C_VEL
LIN {X 0,Y 743.964,Z 399.551,A -85,B 0,C 180,E1 35072.338,E2 35072.338} C_VEL
LIN {X 0,Y 743.967,Z 399.55,A -85,B 0,C 180,E1 35069.913,E2 35069.913} C_VEL
LIN {X 0,Y 744.04,Z 399.551,A -85,B 0,C 180,E1 35067.117,E2 35067.117} C_VEL
LIN {X 0,Y 743.957,Z 399.553,A -85,B 0,C 180,E1 35064.317,E2 35064.317} C_VEL
LIN {X 0,Y 743.948,Z 399.553,A -85,B 0,C 180,E1 35061.962,E2 35061.962} C_VEL
LIN {X 0,Y 743.971,Z 399.551,A -85,B 0,C 180,E1 35059.522,E2 35059.522} C_VEL
LIN {X 0,Y 743.963,Z 399.554,A -85,B 0,C 180,E1 35056.421,E2 35056.421} C_VEL
LIN {X 0,Y 743.936,Z 399.554,A -85,B 0,C 180,E1 35054.018,E2 35054.018} C_VEL
LIN {X 0,Y 743.937,Z 399.546,A -85,B 0,C 180,E1 35051.643,E2 35051.643} C_VEL
LIN {X 0,Y 744.036,Z 399.554,A -85,B 0,C 180,E1 35048.873,E2 35048.873} C_VEL
LIN {X 0,Y 743.933,Z 399.557,A -85,B 0,C 180,E1 35046.065,E2 35046.065} C_VEL
LIN {X 0,Y 743.929,Z 399.559,A -85,B 0,C 180,E1 35043.81,E2 35043.81} C_VEL
LIN {X 0,Y 743.962,Z 399.744,A -85,B 0,C 180,E1 35041.607,E2 35041.607} C_VEL
LIN {X 0,Y 745.514,Z 405.244,A -85,B 0,C 180,E1 35041.089,E2 35041.089} C_VEL
LIN {X 0,Y 745.52,Z 413.639,A -85,B 0,C 180,E1 35040.482,E2 35040.482} C_VEL
LIN {X 0,Y 746.471,Z 418.345,A -85,B 0,C 180,E1 35040.368,E2 35040.368} C_VEL
LIN {X 0,Y 746.056,Z 668.838,A -85,B 0,C 180,E1 35037.602,E2 35037.602} C_VEL
LIN {X 0,Y 745.857,Z 802.52,A -85,B 0,C 180,E1 35036.134,E2 35036.134} C_VEL
LIN {X 0,Y 745.725,Z 827.47,A -85,B 0,C 180,E1 35035.726,E2 35035.726} C_VEL
LIN {X 0,Y 745.628,Z 849.012,A -85,B 0,C 180,E1 35035.242,E2 35035.242} C_VEL
LIN {X 0,Y 745.493,Z 871.827,A -85,B 0,C 180,E1 35034.607,E2 35034.607} C_VEL
LIN {X 0,Y 745.321,Z 895.067,A -85,B 0,C 180,E1 35033.802,E2 35033.802} C_VEL
LIN {X 0,Y 745.182,Z 915.165,A -85,B 0,C 180,E1 35032.984,E2 35032.984} C_VEL
LIN {X 0,Y 744.96,Z 938.594,A -85,B 0,C 180,E1 35031.868,E2 35031.868} C_VEL
LIN {X 0,Y 744.818,Z 957.985,A -85,B 0,C 180,E1 35030.799,E2 35030.799} C_VEL
LIN {X 0,Y 744.616,Z 979.29,A -85,B 0,C 180,E1 35029.452,E2 35029.452} C_VEL
LIN {X 0,Y 744.485,Z 997.32,A -85,B 0,C 180,E1 35028.155,E2 35028.155} C_VEL
LIN {X 0,Y 744.34,Z 1015.016,A -85,B 0,C 180,E1 35026.705,E2 35026.705} C_VEL
LIN {X 0,Y 744.243,Z 1030.606,A -85,B 0,C 180,E1 35025.268,E2 35025.268} C_VEL
LIN {X 0,Y 744.132,Z 1045.683,A -85,B 0,C 180,E1 35023.68,E2 35023.68} C_VEL
LIN {X 0,Y 744.068,Z 1058.264,A -85,B 0,C 180,E1 35022.18,E2 35022.18} C_VEL
LIN {X 0,Y 744.01,Z 1071.612,A -85,B 0,C 180,E1 35020.341,E2 35020.341} C_VEL
LIN {X 0,Y 743.949,Z 1081.149,A -85,B 0,C 180,E1 35018.814,E2 35018.814} C_VEL
LIN {X 0,Y 743.923,Z 1090.725,A -85,B 0,C 180,E1 35017.026,E2 35017.026} C_VEL
LIN {X 0,Y 743.909,Z 1098.128,A -85,B 0,C 180,E1 35015.321,E2 35015.321} C_VEL
LIN {X 0,Y 743.904,Z 1103.903,A -85,B 0,C 180,E1 35013.699,E2 35013.699} C_VEL
LIN {X 0,Y 743.918,Z 1109.261,A -85,B 0,C 180,E1 35011.694,E2 35011.694} C_VEL
LIN {X 0,Y 743.92,Z 1112.287,A -85,B 0,C 180,E1 35010,E2 35010} C_VEL
LIN {X 0,Y 743.915,Z 1114.183,A -85,B 0,C 180,E1 35008.074,E2 35008.074} C_VEL
LIN {X 0,Y 743.89,Z 1114.318,A -85,B 0,C 180,E1 35006.301,E2 35006.301} C_VEL
LIN {X 0,Y 743.906,Z 1113.055,A -85,B 0,C 180,E1 35004.446,E2 35004.446} C_VEL
LIN {X 0,Y 743.894,Z 1110.022,A -85,B 0,C 180,E1 35002.586,E2 35002.586} C_VEL
LIN {X 0,Y 743.907,Z 1106.317,A -85,B 0,C 180,E1 35001.03,E2 35001.03} C_VEL
LIN {X 0,Y 743.914,Z 1100.03,A -85,B 0,C 180,E1 34999.075,E2 34999.075} C_VEL
LIN {X 0,Y 743.917,Z 1093.174,A -85,B 0,C 180,E1 34997.423,E2 34997.423} C_VEL
LIN {X 0,Y 743.96,Z 1084.639,A -85,B 0,C 180,E1 34995.705,E2 34995.705} C_VEL
LIN {X 0,Y 743.987,Z 1073.972,A -85,B 0,C 180,E1 34993.927,E2 34993.927} C_VEL
LIN {X 0,Y 744.038,Z 1063.369,A -85,B 0,C 180,E1 34992.4,E2 34992.4} C_VEL
LIN {X 0,Y 744.111,Z 1049.076,A -85,B 0,C 180,E1 34990.615,E2 34990.615} C_VEL
LIN {X 0,Y 744.184,Z 1035.535,A -85,B 0,C 180,E1 34989.142,E2 34989.142} C_VEL
LIN {X 0,Y 744.329,Z 1018.251,A -85,B 0,C 180,E1 34987.489,E2 34987.489} C_VEL
LIN {X 0,Y 744.434,Z 1001.881,A -85,B 0,C 180,E1 34986.111,E2 34986.111} C_VEL
LIN {X 0,Y 744.598,Z 983.117,A -85,B 0,C 180,E1 34984.721,E2 34984.721} C_VEL
LIN {X 0,Y 744.729,Z 964.944,A -85,B 0,C 180,E1 34983.528,E2 34983.528} C_VEL
LIN {X 0,Y 744.937,Z 943.185,A -85,B 0,C 180,E1 34982.284,E2 34982.284} C_VEL
LIN {X 0,Y 745.085,Z 923.181,A -85,B 0,C 180,E1 34981.286,E2 34981.286} C_VEL
LIN {X 0,Y 745.303,Z 899.623,A -85,B 0,C 180,E1 34980.283,E2 34980.283} C_VEL
LIN {X 0,Y 745.413,Z 878.842,A -85,B 0,C 180,E1 34979.533,E2 34979.533} C_VEL
LIN {X 0,Y 745.622,Z 854.681,A -85,B 0,C 180,E1 34978.811,E2 34978.811} C_VEL
LIN {X 0,Y 745.71,Z 833,A -85,B 0,C 180,E1 34978.299,E2 34978.299} C_VEL
LIN {X 0,Y 745.812,Z 811.88,A -85,B 0,C 180,E1 34977.911,E2 34977.911} C_VEL
LIN {X 0,Y 745.888,Z 780.846,A -85,B 0,C 180,E1 34977.521,E2 34977.521} C_VEL
LIN {X 0,Y 746.28,Z 529.36,A -85,B 0,C 180,E1 34974.778,E2 34974.778} C_VEL
LIN {X 0,Y 746.275,Z 416.642,A -85,B 0,C 180,E1 34973.513,E2 34973.513} C_VEL
LIN {X 0,Y 745.492,Z 413.193,A -85,B 0,C 180,E1 34973.403,E2 34973.403} C_VEL
LIN {X 0,Y 745.299,Z 403.893,A -85,B 0,C 180,E1 34972.709,E2 34972.709} C_VEL
LIN {X 0,Y 743.951,Z 399.712,A -85,B 0,C 180,E1 34972.299,E2 34972.299} C_VEL
LIN {X 0,Y 743.925,Z 399.56,A -85,B 0,C 180,E1 34970.124,E2 34970.124} C_VEL
LIN {X 0,Y 743.939,Z 399.557,A -85,B 0,C 180,E1 34967.776,E2 34967.776} C_VEL
LIN {X 0,Y 744.021,Z 399.555,A -85,B 0,C 180,E1 34964.908,E2 34964.908} C_VEL
LIN {X 0,Y 743.942,Z 399.549,A -85,B 0,C 180,E1 34962.22,E2 34962.22} C_VEL
LIN {X 0,Y 743.941,Z 399.553,A -85,B 0,C 180,E1 34959.874,E2 34959.874} C_VEL
LIN {X 0,Y 743.965,Z 399.554,A -85,B 0,C 180,E1 34957.505,E2 34957.505} C_VEL
LIN {X 0,Y 743.998,Z 399.55,A -85,B 0,C 180,E1 34954.529,E2 34954.529} C_VEL
LIN {X 0,Y 743.955,Z 399.552,A -85,B 0,C 180,E1 34951.975,E2 34951.975} C_VEL
LIN {X 0,Y 743.963,Z 399.546,A -85,B 0,C 180,E1 34949.555,E2 34949.555} C_VEL
LIN {X 0,Y 744.04,Z 399.551,A -85,B 0,C 180,E1 34946.756,E2 34946.756} C_VEL
LIN {X 0,Y 743.971,Z 399.548,A -85,B 0,C 180,E1 34943.947,E2 34943.947} C_VEL
LIN {X 0,Y 743.974,Z 399.553,A -85,B 0,C 180,E1 34941.442,E2 34941.442} C_VEL
LIN {X 0,Y 744.038,Z 399.549,A -85,B 0,C 180,E1 34938.572,E2 34938.572} C_VEL
LIN {X 0,Y 743.978,Z 399.547,A -85,B 0,C 180,E1 34935.753,E2 34935.753} C_VEL
LIN {X 0,Y 744.001,Z 399.553,A -85,B 0,C 180,E1 34933.128,E2 34933.128} C_VEL
LIN {X 0,Y 744.018,Z 399.545,A -85,B 0,C 180,E1 34930.062,E2 34930.062} C_VEL
LIN {X 0,Y 743.988,Z 399.55,A -85,B 0,C 180,E1 34927.321,E2 34927.321} C_VEL
LIN {X 0,Y 744.032,Z 399.551,A -85,B 0,C 180,E1 34924.548,E2 34924.548} C_VEL
LIN {X 0,Y 744.004,Z 399.543,A -85,B 0,C 180,E1 34921.694,E2 34921.694} C_VEL
LIN {X 0,Y 744.025,Z 399.554,A -85,B 0,C 180,E1 34918.845,E2 34918.845} C_VEL
LIN {X 0,Y 744.024,Z 399.543,A -85,B 0,C 180,E1 34915.761,E2 34915.761} C_VEL
LIN {X 0,Y 744.025,Z 399.553,A -85,B 0,C 180,E1 34912.82,E2 34912.82} C_VEL
LIN {X 0,Y 744.036,Z 399.542,A -85,B 0,C 180,E1 34909.782,E2 34909.782} C_VEL
LIN {X 0,Y 744.024,Z 399.551,A -85,B 0,C 180,E1 34906.793,E2 34906.793} C_VEL
LIN {X 0,Y 744.022,Z 399.543,A -85,B 0,C 180,E1 34903.848,E2 34903.848} C_VEL
LIN {X 0,Y 744.014,Z 399.549,A -85,B 0,C 180,E1 34901.021,E2 34901.021} C_VEL
LIN {X 0,Y 744.014,Z 399.549,A -85,B 0,C 180,E1 34898.225,E2 34898.225} C_VEL
LIN {X 0,Y 744.035,Z 399.543,A -85,B 0,C 180,E1 34895.38,E2 34895.38} C_VEL
LIN {X 0,Y 744.026,Z 399.554,A -85,B 0,C 180,E1 34892.377,E2 34892.377} C_VEL
LIN {X 0,Y 744.034,Z 399.541,A -85,B 0,C 180,E1 34889.381,E2 34889.381} C_VEL
LIN {X 0,Y 744.02,Z 399.553,A -85,B 0,C 180,E1 34886.287,E2 34886.287} C_VEL
LIN {X 0,Y 744.019,Z 399.544,A -85,B 0,C 180,E1 34883.366,E2 34883.366} C_VEL
LIN {X 0,Y 744.026,Z 399.555,A -85,B 0,C 180,E1 34880.331,E2 34880.331} C_VEL
LIN {X 0,Y 743.993,Z 399.546,A -85,B 0,C 180,E1 34877.547,E2 34877.547} C_VEL
LIN {X 0,Y 744.031,Z 399.55,A -85,B 0,C 180,E1 34874.69,E2 34874.69} C_VEL
LIN {X 0,Y 743.988,Z 399.554,A -85,B 0,C 180,E1 34871.879,E2 34871.879} C_VEL
LIN {X 0,Y 743.991,Z 399.55,A -85,B 0,C 180,E1 34869.272,E2 34869.272} C_VEL
LIN {X 0,Y 744.017,Z 399.763,A -85,B 0,C 180,E1 34867.262,E2 34867.262} C_VEL
LIN {X 0,Y 745.898,Z 405.719,A -85,B 0,C 180,E1 34866.713,E2 34866.713} C_VEL
LIN {X 0,Y 745.573,Z 441.565,A -85,B 0,C 180,E1 34864.282,E2 34864.282} C_VEL
LIN {X 0,Y 745.639,Z 453.361,A -85,B 0,C 180,E1 34863.515,E2 34863.515} C_VEL
LIN {X 0,Y 746.469,Z 457.681,A -85,B 0,C 180,E1 34863.42,E2 34863.42} C_VEL
LIN {X 0,Y 746.045,Z 710.843,A -85,B 0,C 180,E1 34860.625,E2 34860.625} C_VEL
LIN {X 0,Y 745.867,Z 842.515,A -85,B 0,C 180,E1 34859.179,E2 34859.179} C_VEL
LIN {X 0,Y 745.721,Z 867.473,A -85,B 0,C 180,E1 34858.771,E2 34858.771} C_VEL
LIN {X 0,Y 745.622,Z 888.919,A -85,B 0,C 180,E1 34858.289,E2 34858.289} C_VEL
LIN {X 0,Y 745.498,Z 911.074,A -85,B 0,C 180,E1 34857.674,E2 34857.674} C_VEL
LIN {X 0,Y 745.321,Z 934.807,A -85,B 0,C 180,E1 34856.857,E2 34856.857} C_VEL
LIN {X 0,Y 745.177,Z 955.231,A -85,B 0,C 180,E1 34856.026,E2 34856.026} C_VEL
LIN {X 0,Y 744.964,Z 978.331,A -85,B 0,C 180,E1 34854.926,E2 34854.926} C_VEL
LIN {X 0,Y 744.817,Z 997.354,A -85,B 0,C 180,E1 34853.88,E2 34853.88} C_VEL
LIN {X 0,Y 744.62,Z 1019.23,A -85,B 0,C 180,E1 34852.501,E2 34852.501} C_VEL
LIN {X 0,Y 744.487,Z 1036.823,A -85,B 0,C 180,E1 34851.237,E2 34851.237} C_VEL
LIN {X 0,Y 744.33,Z 1054.602,A -85,B 0,C 180,E1 34849.787,E2 34849.787} C_VEL
LIN {X 0,Y 744.242,Z 1070.494,A -85,B 0,C 180,E1 34848.323,E2 34848.323} C_VEL
LIN {X 0,Y 744.131,Z 1085.799,A -85,B 0,C 180,E1 34846.712,E2 34846.712} C_VEL
LIN {X 0,Y 744.053,Z 1098.533,A -85,B 0,C 180,E1 34845.192,E2 34845.192} C_VEL
LIN {X 0,Y 743.987,Z 1111.752,A -85,B 0,C 180,E1 34843.366,E2 34843.366} C_VEL
LIN {X 0,Y 743.958,Z 1121.101,A -85,B 0,C 180,E1 34841.867,E2 34841.867} C_VEL
LIN {X 0,Y 743.934,Z 1130.759,A -85,B 0,C 180,E1 34840.063,E2 34840.063} C_VEL
LIN {X 0,Y 743.918,Z 1138.206,A -85,B 0,C 180,E1 34838.347,E2 34838.347} C_VEL
LIN {X 0,Y 743.91,Z 1143.997,A -85,B 0,C 180,E1 34836.715,E2 34836.715} C_VEL
LIN {X 0,Y 743.902,Z 1149.178,A -85,B 0,C 180,E1 34834.78,E2 34834.78} C_VEL
LIN {X 0,Y 743.89,Z 1152.121,A -85,B 0,C 180,E1 34833.159,E2 34833.159} C_VEL
LIN {X 0,Y 743.901,Z 1154.032,A -85,B 0,C 180,E1 34831.386,E2 34831.386} C_VEL
LIN {X 0,Y 743.883,Z 1154.373,A -85,B 0,C 180,E1 34829.538,E2 34829.538} C_VEL
LIN {X 0,Y 743.916,Z 1153.43,A -85,B 0,C 180,E1 34827.92,E2 34827.92} C_VEL
LIN {X 0,Y 743.916,Z 1150.605,A -85,B 0,C 180,E1 34825.915,E2 34825.915} C_VEL
LIN {X 0,Y 743.918,Z 1146.687,A -85,B 0,C 180,E1 34824.214,E2 34824.214} C_VEL
LIN {X 0,Y 743.891,Z 1141.2,A -85,B 0,C 180,E1 34822.431,E2 34822.431} C_VEL
LIN {X 0,Y 743.929,Z 1133.737,A -85,B 0,C 180,E1 34820.592,E2 34820.592} C_VEL
LIN {X 0,Y 743.926,Z 1126.333,A -85,B 0,C 180,E1 34819.075,E2 34819.075} C_VEL
LIN {X 0,Y 743.986,Z 1115.909,A -85,B 0,C 180,E1 34817.267,E2 34817.267} C_VEL
LIN {X 0,Y 744.036,Z 1105.097,A -85,B 0,C 180,E1 34815.682,E2 34815.682} C_VEL
LIN {X 0,Y 744.099,Z 1092.116,A -85,B 0,C 180,E1 34814.01,E2 34814.01} C_VEL
LIN {X 0,Y 744.189,Z 1077.619,A -85,B 0,C 180,E1 34812.404,E2 34812.404} C_VEL
LIN {X 0,Y 744.304,Z 1061.99,A -85,B 0,C 180,E1 34810.865,E2 34810.865} C_VEL
LIN {X 0,Y 744.42,Z 1044.831,A -85,B 0,C 180,E1 34809.396,E2 34809.396} C_VEL
LIN {X 0,Y 744.579,Z 1026.474,A -85,B 0,C 180,E1 34807.996,E2 34807.996} C_VEL
LIN {X 0,Y 744.717,Z 1007.739,A -85,B 0,C 180,E1 34806.75,E2 34806.75} C_VEL
LIN {X 0,Y 744.922,Z 987.074,A -85,B 0,C 180,E1 34805.533,E2 34805.533} C_VEL
LIN {X 0,Y 745.071,Z 966.344,A -85,B 0,C 180,E1 34804.483,E2 34804.483} C_VEL
LIN {X 0,Y 745.278,Z 944.262,A -85,B 0,C 180,E1 34803.507,E2 34803.507} C_VEL
LIN {X 0,Y 745.41,Z 921.533,A -85,B 0,C 180,E1 34802.669,E2 34802.669} C_VEL
LIN {X 0,Y 745.547,Z 900.872,A -85,B 0,C 180,E1 34802.026,E2 34802.026} C_VEL
LIN {X 0,Y 745.695,Z 875.927,A -85,B 0,C 180,E1 34801.406,E2 34801.406} C_VEL
LIN {X 0,Y 745.798,Z 855.578,A -85,B 0,C 180,E1 34801.018,E2 34801.018} C_VEL
LIN {X 0,Y 745.883,Z 832.13,A -85,B 0,C 180,E1 34800.689,E2 34800.689} C_VEL
LIN {X 0,Y 746.198,Z 588.481,A -85,B 0,C 180,E1 34798.031,E2 34798.031} C_VEL
LIN {X 0,Y 746.29,Z 455.925,A -85,B 0,C 180,E1 34796.551,E2 34796.551} C_VEL
LIN {X 0,Y 745.556,Z 452.716,A -85,B 0,C 180,E1 34796.458,E2 34796.458} C_VEL
LIN {X 0,Y 745.842,Z 413.943,A -85,B 0,C 180,E1 34793.852,E2 34793.852} C_VEL
LIN {X 0,Y 745.853,Z 404.898,A -85,B 0,C 180,E1 34793.227,E2 34793.227} C_VEL
LIN {X 0,Y 744.009,Z 399.715,A -85,B 0,C 180,E1 34792.728,E2 34792.728} C_VEL
LIN {X 0,Y 743.985,Z 399.552,A -85,B 0,C 180,E1 34790.122,E2 34790.122} C_VEL
LIN {X 0,Y 744.034,Z 399.55,A -85,B 0,C 180,E1 34787.261,E2 34787.261} C_VEL
LIN {X 0,Y 743.989,Z 399.549,A -85,B 0,C 180,E1 34784.444,E2 34784.444} C_VEL
LIN {X 0,Y 744.03,Z 399.546,A -85,B 0,C 180,E1 34781.651,E2 34781.651} C_VEL
LIN {X 0,Y 744.017,Z 399.545,A -85,B 0,C 180,E1 34778.665,E2 34778.665} C_VEL
LIN {X 0,Y 744.013,Z 399.551,A -85,B 0,C 180,E1 34775.775,E2 34775.775} C_VEL
LIN {X 0,Y 744.037,Z 399.541,A -85,B 0,C 180,E1 34772.791,E2 34772.791} C_VEL
LIN {X 0,Y 744.004,Z 399.551,A -85,B 0,C 180,E1 34769.906,E2 34769.906} C_VEL
LIN {X 0,Y 744.021,Z 399.55,A -85,B 0,C 180,E1 34767.103,E2 34767.103} C_VEL
LIN {X 0,Y 744.017,Z 399.542,A -85,B 0,C 180,E1 34764.283,E2 34764.283} C_VEL
LIN {X 0,Y 744.034,Z 399.554,A -85,B 0,C 180,E1 34761.358,E2 34761.358} C_VEL
LIN {X 0,Y 744.031,Z 399.541,A -85,B 0,C 180,E1 34758.329,E2 34758.329} C_VEL
LIN {X 0,Y 744.038,Z 399.553,A -85,B 0,C 180,E1 34755.352,E2 34755.352} C_VEL
LIN {X 0,Y 744.035,Z 399.542,A -85,B 0,C 180,E1 34752.312,E2 34752.312} C_VEL
LIN {X 0,Y 744.033,Z 399.552,A -85,B 0,C 180,E1 34749.28,E2 34749.28} C_VEL
LIN {X 0,Y 744.021,Z 399.544,A -85,B 0,C 180,E1 34746.327,E2 34746.327} C_VEL
LIN {X 0,Y 744.036,Z 399.552,A -85,B 0,C 180,E1 34743.313,E2 34743.313} C_VEL
LIN {X 0,Y 744,Z 399.547,A -85,B 0,C 180,E1 34740.462,E2 34740.462} C_VEL
LIN {X 0,Y 744.027,Z 399.547,A -85,B 0,C 180,E1 34737.612,E2 34737.612} C_VEL
LIN {X 0,Y 743.995,Z 399.551,A -85,B 0,C 180,E1 34734.756,E2 34734.756} C_VEL
LIN {X 0,Y 744.021,Z 399.542,A -85,B 0,C 180,E1 34731.966,E2 34731.966} C_VEL
LIN {X 0,Y 744.033,Z 399.542,A -85,B 0,C 180,E1 34731.802,E2 34731.802} C_VEL
LIN {X 0,Y 743.058,Z 399.674,A -85,B 0,C 180,E1 34731.209,E2 34731.209} C_VEL
LIN {X 0,Y 736.64,Z 400.484,A -85,B 0,C 180,E1 34729.549,E2 34729.549} C_VEL
LIN {X 0,Y 736.091,Z 400.544,A -85,B 0,C 180,E1 34729.117,E2 34729.117} C_VEL
LIN {X 0,Y 736.042,Z 400.535,A -85,B 0,C 180,E1 34726.407,E2 34726.407} C_VEL
LIN {X 0,Y 736.093,Z 400.534,A -85,B 0,C 180,E1 34723.669,E2 34723.669} C_VEL
LIN {X 0,Y 736.053,Z 400.54,A -85,B 0,C 180,E1 34720.725,E2 34720.725} C_VEL
LIN {X 0,Y 736.035,Z 400.539,A -85,B 0,C 180,E1 34718.102,E2 34718.102} C_VEL
LIN {X 0,Y 736.099,Z 400.534,A -85,B 0,C 180,E1 34715.333,E2 34715.333} C_VEL
LIN {X 0,Y 736.033,Z 400.54,A -85,B 0,C 180,E1 34712.491,E2 34712.491} C_VEL
LIN {X 0,Y 736.024,Z 400.54,A -85,B 0,C 180,E1 34710.005,E2 34710.005} C_VEL
LIN {X 0,Y 736.1,Z 400.538,A -85,B 0,C 180,E1 34707.228,E2 34707.228} C_VEL
LIN {X 0,Y 736.021,Z 400.542,A -85,B 0,C 180,E1 34704.352,E2 34704.352} C_VEL
LIN {X 0,Y 736.01,Z 400.542,A -85,B 0,C 180,E1 34701.994,E2 34701.994} C_VEL
LIN {X 0,Y 736.034,Z 400.54,A -85,B 0,C 180,E1 34699.507,E2 34699.507} C_VEL
LIN {X 0,Y 736.03,Z 400.543,A -85,B 0,C 180,E1 34696.468,E2 34696.468} C_VEL
LIN {X 0,Y 735.998,Z 400.543,A -85,B 0,C 180,E1 34694.055,E2 34694.055} C_VEL
LIN {X 0,Y 735.994,Z 400.533,A -85,B 0,C 180,E1 34691.736,E2 34691.736} C_VEL
LIN {X 0,Y 736.047,Z 400.546,A -85,B 0,C 180,E1 34689.133,E2 34689.133} C_VEL
LIN {X 0,Y 736.004,Z 400.547,A -85,B 0,C 180,E1 34686.198,E2 34686.198} C_VEL
LIN {X 0,Y 735.992,Z 400.55,A -85,B 0,C 180,E1 34683.85,E2 34683.85} C_VEL
LIN {X 0,Y 736.034,Z 400.795,A -85,B 0,C 180,E1 34681.947,E2 34681.947} C_VEL
LIN {X 0,Y 738.322,Z 408.213,A -85,B 0,C 180,E1 34681.244,E2 34681.244} C_VEL
LIN {X 0,Y 738.362,Z 413.848,A -85,B 0,C 180,E1 34680.844,E2 34680.844} C_VEL
LIN {X 0,Y 739.782,Z 420.18,A -85,B 0,C 180,E1 34680.689,E2 34680.689} C_VEL
LIN {X 0,Y 739.161,Z 671.591,A -85,B 0,C 180,E1 34677.889,E2 34677.889} C_VEL
LIN {X 0,Y 738.861,Z 802.655,A -85,B 0,C 180,E1 34676.436,E2 34676.436} C_VEL
LIN {X 0,Y 738.667,Z 827.876,A -85,B 0,C 180,E1 34676.019,E2 34676.019} C_VEL
LIN {X 0,Y 738.515,Z 849.41,A -85,B 0,C 180,E1 34675.529,E2 34675.529} C_VEL
LIN {X 0,Y 738.318,Z 872.452,A -85,B 0,C 180,E1 34674.881,E2 34674.881} C_VEL
LIN {X 0,Y 738.043,Z 895.634,A -85,B 0,C 180,E1 34674.066,E2 34674.066} C_VEL
LIN {X 0,Y 737.827,Z 916.984,A -85,B 0,C 180,E1 34673.184,E2 34673.184} C_VEL
LIN {X 0,Y 737.5,Z 939.284,A -85,B 0,C 180,E1 34672.1,E2 34672.1} C_VEL
LIN {X 0,Y 737.28,Z 959.323,A -85,B 0,C 180,E1 34670.98,E2 34670.98} C_VEL
LIN {X 0,Y 736.98,Z 979.812,A -85,B 0,C 180,E1 34669.662,E2 34669.662} C_VEL
LIN {X 0,Y 736.782,Z 998.4,A -85,B 0,C 180,E1 34668.306,E2 34668.306} C_VEL
LIN {X 0,Y 736.558,Z 1015.805,A -85,B 0,C 180,E1 34666.852,E2 34666.852} C_VEL
LIN {X 0,Y 736.411,Z 1031.803,A -85,B 0,C 180,E1 34665.353,E2 34665.353} C_VEL
LIN {X 0,Y 736.243,Z 1046.687,A -85,B 0,C 180,E1 34663.749,E2 34663.749} C_VEL
LIN {X 0,Y 736.14,Z 1060.43,A -85,B 0,C 180,E1 34662.074,E2 34662.074} C_VEL
LIN {X 0,Y 736.054,Z 1072.645,A -85,B 0,C 180,E1 34660.33,E2 34660.33} C_VEL
LIN {X 0,Y 735.986,Z 1082.723,A -85,B 0,C 180,E1 34658.673,E2 34658.673} C_VEL
LIN {X 0,Y 735.923,Z 1092.286,A -85,B 0,C 180,E1 34656.789,E2 34656.789} C_VEL
LIN {X 0,Y 735.928,Z 1099.031,A -85,B 0,C 180,E1 34655.179,E2 34655.179} C_VEL
LIN {X 0,Y 735.889,Z 1105.457,A -85,B 0,C 180,E1 34653.272,E2 34653.272} C_VEL
LIN {X 0,Y 735.913,Z 1109.645,A -85,B 0,C 180,E1 34651.557,E2 34651.557} C_VEL
LIN {X 0,Y 735.91,Z 1112.56,A -85,B 0,C 180,E1 34649.844,E2 34649.844} C_VEL
LIN {X 0,Y 735.906,Z 1114.259,A -85,B 0,C 180,E1 34647.82,E2 34647.82} C_VEL
LIN {X 0,Y 735.897,Z 1114.286,A -85,B 0,C 180,E1 34646.183,E2 34646.183} C_VEL
LIN {X 0,Y 735.902,Z 1112.796,A -85,B 0,C 180,E1 34644.229,E2 34644.229} C_VEL
LIN {X 0,Y 735.908,Z 1109.795,A -85,B 0,C 180,E1 34642.427,E2 34642.427} C_VEL
LIN {X 0,Y 735.889,Z 1105.606,A -85,B 0,C 180,E1 34640.695,E2 34640.695} C_VEL
LIN {X 0,Y 735.93,Z 1099.286,A -85,B 0,C 180,E1 34638.797,E2 34638.797} C_VEL
LIN {X 0,Y 735.923,Z 1092.661,A -85,B 0,C 180,E1 34637.205,E2 34637.205} C_VEL
LIN {X 0,Y 735.995,Z 1083.454,A -85,B 0,C 180,E1 34635.363,E2 34635.363} C_VEL
LIN {X 0,Y 736.044,Z 1073.218,A -85,B 0,C 180,E1 34633.668,E2 34633.668} C_VEL
LIN {X 0,Y 736.129,Z 1061.35,A -85,B 0,C 180,E1 34631.959,E2 34631.959} C_VEL
LIN {X 0,Y 736.242,Z 1047.328,A -85,B 0,C 180,E1 34630.235,E2 34630.235} C_VEL
LIN {X 0,Y 736.389,Z 1032.816,A -85,B 0,C 180,E1 34628.66,E2 34628.66} C_VEL
LIN {X 0,Y 736.557,Z 1016.412,A -85,B 0,C 180,E1 34627.112,E2 34627.112} C_VEL
LIN {X 0,Y 736.779,Z 998.801,A -85,B 0,C 180,E1 34625.634,E2 34625.634} C_VEL
LIN {X 0,Y 736.978,Z 980.105,A -85,B 0,C 180,E1 34624.268,E2 34624.268} C_VEL
LIN {X 0,Y 737.283,Z 959.399,A -85,B 0,C 180,E1 34622.935,E2 34622.935} C_VEL
LIN {X 0,Y 737.498,Z 940,A -85,B 0,C 180,E1 34621.848,E2 34621.848} C_VEL
LIN {X 0,Y 737.82,Z 918.227,A -85,B 0,C 180,E1 34620.78,E2 34620.78} C_VEL
LIN {X 0,Y 738.041,Z 896.33,A -85,B 0,C 180,E1 34619.871,E2 34619.871} C_VEL
LIN {X 0,Y 738.29,Z 873.749,A -85,B 0,C 180,E1 34619.071,E2 34619.071} C_VEL
LIN {X 0,Y 738.519,Z 849.945,A -85,B 0,C 180,E1 34618.395,E2 34618.395} C_VEL
LIN {X 0,Y 738.665,Z 828.861,A -85,B 0,C 180,E1 34617.912,E2 34617.912} C_VEL
LIN {X 0,Y 738.861,Z 803.142,A -85,B 0,C 180,E1 34617.481,E2 34617.481} C_VEL
LIN {X 0,Y 739.076,Z 718.839,A -85,B 0,C 180,E1 34616.54,E2 34616.54} C_VEL
LIN {X 0,Y 739.666,Z 466.282,A -85,B 0,C 180,E1 34613.741,E2 34613.741} C_VEL
LIN {X 0,Y 739.59,Z 418.554,A -85,B 0,C 180,E1 34613.192,E2 34613.192} C_VEL
LIN {X 0,Y 738.301,Z 413.254,A -85,B 0,C 180,E1 34613.036,E2 34613.036} C_VEL
LIN {X 0,Y 738.233,Z 407.365,A -85,B 0,C 180,E1 34612.597,E2 34612.597} C_VEL
LIN {X 0,Y 736.007,Z 400.647,A -85,B 0,C 180,E1 34611.932,E2 34611.932} C_VEL
LIN {X 0,Y 736.043,Z 400.546,A -85,B 0,C 180,E1 34609.405,E2 34609.405} C_VEL
LIN {X 0,Y 736.01,Z 400.546,A -85,B 0,C 180,E1 34606.467,E2 34606.467} C_VEL
LIN {X 0,Y 735.996,Z 400.545,A -85,B 0,C 180,E1 34604.074,E2 34604.074} C_VEL
LIN {X 0,Y 736.005,Z 400.537,A -85,B 0,C 180,E1 34601.735,E2 34601.735} C_VEL
LIN {X 0,Y 736.101,Z 400.54,A -85,B 0,C 180,E1 34598.871,E2 34598.871} C_VEL
LIN {X 0,Y 736.011,Z 400.53,A -85,B 0,C 180,E1 34596.067,E2 34596.067} C_VEL
LIN {X 0,Y 736.016,Z 400.542,A -85,B 0,C 180,E1 34593.661,E2 34593.661} C_VEL
LIN {X 0,Y 736.101,Z 400.532,A -85,B 0,C 180,E1 34590.853,E2 34590.853} C_VEL
LIN {X 0,Y 736.027,Z 400.537,A -85,B 0,C 180,E1 34588.037,E2 34588.037} C_VEL
LIN {X 0,Y 736.028,Z 400.542,A -85,B 0,C 180,E1 34585.572,E2 34585.572} C_VEL
LIN {X 0,Y 736.101,Z 400.542,A -85,B 0,C 180,E1 34582.776,E2 34582.776} C_VEL
LIN {X 0,Y 736.041,Z 400.536,A -85,B 0,C 180,E1 34579.937,E2 34579.937} C_VEL
LIN {X 0,Y 736.048,Z 400.542,A -85,B 0,C 180,E1 34577.308,E2 34577.308} C_VEL
LIN {X 0,Y 736.101,Z 400.535,A -85,B 0,C 180,E1 34574.394,E2 34574.394} C_VEL
LIN {X 0,Y 736.043,Z 400.536,A -85,B 0,C 180,E1 34571.599,E2 34571.599} C_VEL
LIN {X 0,Y 736.095,Z 400.544,A -85,B 0,C 180,E1 34568.83,E2 34568.83} C_VEL
LIN {X 0,Y 736.067,Z 400.533,A -85,B 0,C 180,E1 34565.848,E2 34565.848} C_VEL
LIN {X 0,Y 736.069,Z 400.541,A -85,B 0,C 180,E1 34563.037,E2 34563.037} C_VEL
LIN {X 0,Y 736.103,Z 400.531,A -85,B 0,C 180,E1 34560,E2 34560} C_VEL
LIN {X 0,Y 736.063,Z 400.537,A -85,B 0,C 180,E1 34557.119,E2 34557.119} C_VEL
LIN {X 0,Y 736.085,Z 400.537,A -85,B 0,C 180,E1 34554.309,E2 34554.309} C_VEL
LIN {X 0,Y 736.071,Z 400.533,A -85,B 0,C 180,E1 34551.467,E2 34551.467} C_VEL
LIN {X 0,Y 736.094,Z 400.54,A -85,B 0,C 180,E1 34548.561,E2 34548.561} C_VEL
LIN {X 0,Y 736.087,Z 400.533,A -85,B 0,C 180,E1 34545.526,E2 34545.526} C_VEL
LIN {X 0,Y 736.095,Z 400.543,A -85,B 0,C 180,E1 34542.53,E2 34542.53} C_VEL
LIN {X 0,Y 736.094,Z 400.53,A -85,B 0,C 180,E1 34539.484,E2 34539.484} C_VEL
LIN {X 0,Y 736.091,Z 400.544,A -85,B 0,C 180,E1 34536.461,E2 34536.461} C_VEL
LIN {X 0,Y 736.093,Z 400.528,A -85,B 0,C 180,E1 34533.455,E2 34533.455} C_VEL
LIN {X 0,Y 736.086,Z 400.542,A -85,B 0,C 180,E1 34530.366,E2 34530.366} C_VEL
LIN {X 0,Y 736.088,Z 400.532,A -85,B 0,C 180,E1 34527.373,E2 34527.373} C_VEL
LIN {X 0,Y 736.085,Z 400.542,A -85,B 0,C 180,E1 34524.323,E2 34524.323} C_VEL
LIN {X 0,Y 736.069,Z 400.534,A -85,B 0,C 180,E1 34521.427,E2 34521.427} C_VEL
LIN {X 0,Y 736.094,Z 400.541,A -85,B 0,C 180,E1 34518.375,E2 34518.375} C_VEL
LIN {X 0,Y 736.05,Z 400.538,A -85,B 0,C 180,E1 34515.604,E2 34515.604} C_VEL
LIN {X 0,Y 736.096,Z 400.538,A -85,B 0,C 180,E1 34512.78,E2 34512.78} C_VEL
LIN {X 0,Y 736.046,Z 400.54,A -85,B 0,C 180,E1 34509.867,E2 34509.867} C_VEL
LIN {X 0,Y 736.073,Z 400.773,A -85,B 0,C 180,E1 34507.661,E2 34507.661} C_VEL
LIN {X 0,Y 738.896,Z 408.94,A -85,B 0,C 180,E1 34506.893,E2 34506.893} C_VEL
LIN {X 0,Y 738.446,Z 445.017,A -85,B 0,C 180,E1 34504.424,E2 34504.424} C_VEL
LIN {X 0,Y 738.515,Z 453.466,A -85,B 0,C 180,E1 34503.879,E2 34503.879} C_VEL
LIN {X 0,Y 739.783,Z 459.404,A -85,B 0,C 180,E1 34503.743,E2 34503.743} C_VEL
LIN {X 0,Y 739.152,Z 712.362,A -85,B 0,C 180,E1 34500.925,E2 34500.925} C_VEL
LIN {X 0,Y 738.87,Z 842.623,A -85,B 0,C 180,E1 34499.481,E2 34499.481} C_VEL
LIN {X 0,Y 738.664,Z 867.848,A -85,B 0,C 180,E1 34499.064,E2 34499.064} C_VEL
LIN {X 0,Y 738.509,Z 889.354,A -85,B 0,C 180,E1 34498.576,E2 34498.576} C_VEL
LIN {X 0,Y 738.318,Z 912.614,A -85,B 0,C 180,E1 34497.92,E2 34497.92} C_VEL
LIN {X 0,Y 738.045,Z 935.538,A -85,B 0,C 180,E1 34497.115,E2 34497.115} C_VEL
LIN {X 0,Y 737.827,Z 956.229,A -85,B 0,C 180,E1 34496.262,E2 34496.262} C_VEL
LIN {X 0,Y 737.505,Z 979.137,A -85,B 0,C 180,E1 34495.153,E2 34495.153} C_VEL
LIN {X 0,Y 737.28,Z 998.883,A -85,B 0,C 180,E1 34494.05,E2 34494.05} C_VEL
LIN {X 0,Y 736.993,Z 1019.232,A -85,B 0,C 180,E1 34492.747,E2 34492.747} C_VEL
LIN {X 0,Y 736.789,Z 1037.104,A -85,B 0,C 180,E1 34491.449,E2 34491.449} C_VEL
LIN {X 0,Y 736.563,Z 1054.602,A -85,B 0,C 180,E1 34490.005,E2 34490.005} C_VEL
LIN {X 0,Y 736.424,Z 1070.493,A -85,B 0,C 180,E1 34488.525,E2 34488.525} C_VEL
LIN {X 0,Y 736.241,Z 1085.801,A -85,B 0,C 180,E1 34486.896,E2 34486.896} C_VEL
LIN {X 0,Y 736.14,Z 1098.715,A -85,B 0,C 180,E1 34485.336,E2 34485.336} C_VEL
LIN {X 0,Y 736.044,Z 1111.753,A -85,B 0,C 180,E1 34483.512,E2 34483.512} C_VEL
LIN {X 0,Y 735.992,Z 1121.12,A -85,B 0,C 180,E1 34481.994,E2 34481.994} C_VEL
LIN {X 0,Y 735.959,Z 1130.76,A -85,B 0,C 180,E1 34480.173,E2 34480.173} C_VEL
LIN {X 0,Y 735.92,Z 1138.206,A -85,B 0,C 180,E1 34478.438,E2 34478.438} C_VEL
LIN {X 0,Y 735.917,Z 1143.997,A -85,B 0,C 180,E1 34476.789,E2 34476.789} C_VEL
LIN {X 0,Y 735.898,Z 1149.178,A -85,B 0,C 180,E1 34474.832,E2 34474.832} C_VEL
LIN {X 0,Y 735.892,Z 1152.122,A -85,B 0,C 180,E1 34473.194,E2 34473.194} C_VEL
LIN {X 0,Y 735.905,Z 1154.099,A -85,B 0,C 180,E1 34471.324,E2 34471.324} C_VEL
LIN {X 0,Y 735.881,Z 1154.351,A -85,B 0,C 180,E1 34469.455,E2 34469.455} C_VEL
LIN {X 0,Y 735.917,Z 1153.297,A -85,B 0,C 180,E1 34467.742,E2 34467.742} C_VEL
LIN {X 0,Y 735.915,Z 1150.288,A -85,B 0,C 180,E1 34465.714,E2 34465.714} C_VEL
LIN {X 0,Y 735.923,Z 1146.353,A -85,B 0,C 180,E1 34464.024,E2 34464.024} C_VEL
LIN {X 0,Y 735.915,Z 1140.271,A -85,B 0,C 180,E1 34462.096,E2 34462.096} C_VEL
LIN {X 0,Y 735.932,Z 1133.245,A -85,B 0,C 180,E1 34460.38,E2 34460.38} C_VEL
LIN {X 0,Y 735.966,Z 1125.11,A -85,B 0,C 180,E1 34458.718,E2 34458.718} C_VEL
LIN {X 0,Y 736.02,Z 1114.352,A -85,B 0,C 180,E1 34456.887,E2 34456.887} C_VEL
LIN {X 0,Y 736.109,Z 1103.953,A -85,B 0,C 180,E1 34455.365,E2 34455.365} C_VEL
LIN {X 0,Y 736.227,Z 1090.044,A -85,B 0,C 180,E1 34453.591,E2 34453.591} C_VEL
LIN {X 0,Y 736.329,Z 1076.067,A -85,B 0,C 180,E1 34452.046,E2 34452.046} C_VEL
LIN {X 0,Y 736.53,Z 1059.246,A -85,B 0,C 180,E1 34450.408,E2 34450.408} C_VEL
LIN {X 0,Y 736.711,Z 1042.805,A -85,B 0,C 180,E1 34449.003,E2 34449.003} C_VEL
LIN {X 0,Y 736.963,Z 1022.854,A -85,B 0,C 180,E1 34447.504,E2 34447.504} C_VEL
LIN {X 0,Y 737.195,Z 1004.357,A -85,B 0,C 180,E1 34446.282,E2 34446.282} C_VEL
LIN {X 0,Y 737.48,Z 982.344,A -85,B 0,C 180,E1 34445.018,E2 34445.018} C_VEL
LIN {X 0,Y 737.72,Z 962.785,A -85,B 0,C 180,E1 34444.037,E2 34444.037} C_VEL
LIN {X 0,Y 738.022,Z 939.382,A -85,B 0,C 180,E1 34443.034,E2 34443.034} C_VEL
LIN {X 0,Y 738.199,Z 919.691,A -85,B 0,C 180,E1 34442.316,E2 34442.316} C_VEL
LIN {X 0,Y 738.492,Z 896.035,A -85,B 0,C 180,E1 34441.594,E2 34441.594} C_VEL
LIN {X 0,Y 738.638,Z 873.309,A -85,B 0,C 180,E1 34441.051,E2 34441.051} C_VEL
LIN {X 0,Y 738.792,Z 852.207,A -85,B 0,C 180,E1 34440.658,E2 34440.658} C_VEL
LIN {X 0,Y 738.923,Z 821.027,A -85,B 0,C 180,E1 34440.263,E2 34440.263} C_VEL
LIN {X 0,Y 739.409,Z 584.865,A -85,B 0,C 180,E1 34437.662,E2 34437.662} C_VEL
LIN {X 0,Y 739.606,Z 457.78,A -85,B 0,C 180,E1 34436.229,E2 34436.229} C_VEL
LIN {X 0,Y 738.414,Z 452.716,A -85,B 0,C 180,E1 34436.09,E2 34436.09} C_VEL
LIN {X 0,Y 738.83,Z 415.324,A -85,B 0,C 180,E1 34433.55,E2 34433.55} C_VEL
LIN {X 0,Y 738.893,Z 408.418,A -85,B 0,C 180,E1 34433.07,E2 34433.07} C_VEL
LIN {X 0,Y 736.064,Z 400.714,A -85,B 0,C 180,E1 34432.328,E2 34432.328} C_VEL
LIN {X 0,Y 736.102,Z 400.539,A -85,B 0,C 180,E1 34429.613,E2 34429.613} C_VEL
LIN {X 0,Y 736.06,Z 400.538,A -85,B 0,C 180,E1 34426.685,E2 34426.685} C_VEL
LIN {X 0,Y 736.062,Z 400.543,A -85,B 0,C 180,E1 34423.948,E2 34423.948} C_VEL
LIN {X 0,Y 736.094,Z 400.528,A -85,B 0,C 180,E1 34420.952,E2 34420.952} C_VEL
LIN {X 0,Y 736.055,Z 400.54,A -85,B 0,C 180,E1 34418.136,E2 34418.136} C_VEL
LIN {X 0,Y 736.092,Z 400.542,A -85,B 0,C 180,E1 34415.357,E2 34415.357} C_VEL
LIN {X 0,Y 736.073,Z 400.532,A -85,B 0,C 180,E1 34412.451,E2 34412.451} C_VEL
LIN {X 0,Y 736.094,Z 400.543,A -85,B 0,C 180,E1 34409.544,E2 34409.544} C_VEL
LIN {X 0,Y 736.088,Z 400.532,A -85,B 0,C 180,E1 34406.459,E2 34406.459} C_VEL
LIN {X 0,Y 736.095,Z 400.54,A -85,B 0,C 180,E1 34403.453,E2 34403.453} C_VEL
LIN {X 0,Y 736.094,Z 400.531,A -85,B 0,C 180,E1 34400.4,E2 34400.4} C_VEL
LIN {X 0,Y 736.097,Z 400.543,A -85,B 0,C 180,E1 34397.388,E2 34397.388} C_VEL
LIN {X 0,Y 736.1,Z 400.527,A -85,B 0,C 180,E1 34394.313,E2 34394.313} C_VEL
LIN {X 0,Y 736.092,Z 400.543,A -85,B 0,C 180,E1 34391.259,E2 34391.259} C_VEL
LIN {X 0,Y 736.09,Z 400.528,A -85,B 0,C 180,E1 34388.279,E2 34388.279} C_VEL
LIN {X 0,Y 736.094,Z 400.542,A -85,B 0,C 180,E1 34385.222,E2 34385.222} C_VEL
LIN {X 0,Y 736.078,Z 400.531,A -85,B 0,C 180,E1 34382.258,E2 34382.258} C_VEL
LIN {X 0,Y 736.094,Z 400.543,A -85,B 0,C 180,E1 34379.222,E2 34379.222} C_VEL
LIN {X 0,Y 736.06,Z 400.534,A -85,B 0,C 180,E1 34376.339,E2 34376.339} C_VEL
LIN {X 0,Y 736.093,Z 400.539,A -85,B 0,C 180,E1 34373.448,E2 34373.448} C_VEL
LIN {X 0,Y 736.049,Z 400.539,A -85,B 0,C 180,E1 34370.618,E2 34370.618} C_VEL
LIN {X 0,Y 736.091,Z 400.544,A -85,B 0,C 180,E1 34369.117,E2 34369.117} C_VEL
LIN {X 0,Y 735.079,Z 400.661,A -85,B 0,C 180,E1 34368.517,E2 34368.517} C_VEL
LIN {X 0,Y 728.635,Z 401.464,A -85,B 0,C 180,E1 34366.838,E2 34366.838} C_VEL
LIN {X 0,Y 728.103,Z 401.523,A -85,B 0,C 180,E1 34366.402,E2 34366.402} C_VEL
LIN {X 0,Y 728.156,Z 401.523,A -85,B 0,C 180,E1 34363.65,E2 34363.65} C_VEL
LIN {X 0,Y 728.107,Z 401.528,A -85,B 0,C 180,E1 34360.638,E2 34360.638} C_VEL
LIN {X 0,Y 728.098,Z 401.527,A -85,B 0,C 180,E1 34358.066,E2 34358.066} C_VEL
LIN {X 0,Y 728.16,Z 401.525,A -85,B 0,C 180,E1 34355.186,E2 34355.186} C_VEL
LIN {X 0,Y 728.088,Z 401.528,A -85,B 0,C 180,E1 34352.349,E2 34352.349} C_VEL
LIN {X 0,Y 728.096,Z 401.528,A -85,B 0,C 180,E1 34349.826,E2 34349.826} C_VEL
LIN {X 0,Y 728.14,Z 401.531,A -85,B 0,C 180,E1 34346.87,E2 34346.87} C_VEL
LIN {X 0,Y 728.075,Z 401.53,A -85,B 0,C 180,E1 34344.194,E2 34344.194} C_VEL
LIN {X 0,Y 728.079,Z 401.531,A -85,B 0,C 180,E1 34341.771,E2 34341.771} C_VEL
LIN {X 0,Y 728.159,Z 401.52,A -85,B 0,C 180,E1 34338.927,E2 34338.927} C_VEL
LIN {X 0,Y 728.064,Z 401.532,A -85,B 0,C 180,E1 34336.138,E2 34336.138} C_VEL
LIN {X 0,Y 728.06,Z 401.532,A -85,B 0,C 180,E1 34333.803,E2 34333.803} C_VEL
LIN {X 0,Y 728.116,Z 401.518,A -85,B 0,C 180,E1 34331.132,E2 34331.132} C_VEL
LIN {X 0,Y 728.065,Z 401.529,A -85,B 0,C 180,E1 34328.227,E2 34328.227} C_VEL
LIN {X 0,Y 728.05,Z 401.537,A -85,B 0,C 180,E1 34325.875,E2 34325.875} C_VEL
LIN {X 0,Y 728.06,Z 401.54,A -85,B 0,C 180,E1 34323.526,E2 34323.526} C_VEL
LIN {X 0,Y 728.122,Z 401.752,A -85,B 0,C 180,E1 34322.313,E2 34322.313} C_VEL
LIN {X 0,Y 731.136,Z 411.182,A -85,B 0,C 180,E1 34321.403,E2 34321.403} C_VEL
LIN {X 0,Y 731.279,Z 414.261,A -85,B 0,C 180,E1 34321.209,E2 34321.209} C_VEL
LIN {X 0,Y 733.117,Z 421.939,A -85,B 0,C 180,E1 34321.017,E2 34321.017} C_VEL
LIN {X 0,Y 732.288,Z 673.478,A -85,B 0,C 180,E1 34318.19,E2 34318.19} C_VEL
LIN {X 0,Y 731.885,Z 802.79,A -85,B 0,C 180,E1 34316.743,E2 34316.743} C_VEL
LIN {X 0,Y 731.635,Z 828.116,A -85,B 0,C 180,E1 34316.32,E2 34316.32} C_VEL
LIN {X 0,Y 731.422,Z 849.808,A -85,B 0,C 180,E1 34315.822,E2 34315.822} C_VEL
LIN {X 0,Y 731.16,Z 872.708,A -85,B 0,C 180,E1 34315.17,E2 34315.17} C_VEL
LIN {X 0,Y 730.79,Z 895.494,A -85,B 0,C 180,E1 34314.364,E2 34314.364} C_VEL
LIN {X 0,Y 730.488,Z 917.833,A -85,B 0,C 180,E1 34313.431,E2 34313.431} C_VEL
LIN {X 0,Y 730.057,Z 939.974,A -85,B 0,C 180,E1 34312.338,E2 34312.338} C_VEL
LIN {X 0,Y 729.749,Z 960.661,A -85,B 0,C 180,E1 34311.164,E2 34311.164} C_VEL
LIN {X 0,Y 729.352,Z 980.866,A -85,B 0,C 180,E1 34309.839,E2 34309.839} C_VEL
LIN {X 0,Y 729.071,Z 999.842,A -85,B 0,C 180,E1 34308.429,E2 34308.429} C_VEL
LIN {X 0,Y 728.78,Z 1016.713,A -85,B 0,C 180,E1 34306.992,E2 34306.992} C_VEL
LIN {X 0,Y 728.57,Z 1032.931,A -85,B 0,C 180,E1 34305.441,E2 34305.441} C_VEL
LIN {X 0,Y 728.357,Z 1046.993,A -85,B 0,C 180,E1 34303.901,E2 34303.901} C_VEL
LIN {X 0,Y 728.223,Z 1060.7,A -85,B 0,C 180,E1 34302.207,E2 34302.207} C_VEL
LIN {X 0,Y 728.103,Z 1072.87,A -85,B 0,C 180,E1 34300.444,E2 34300.444} C_VEL
LIN {X 0,Y 728.013,Z 1082.919,A -85,B 0,C 180,E1 34298.769,E2 34298.769} C_VEL
LIN {X 0,Y 727.941,Z 1092.086,A -85,B 0,C 180,E1 34296.943,E2 34296.943} C_VEL
LIN {X 0,Y 727.923,Z 1098.69,A -85,B 0,C 180,E1 34295.36,E2 34295.36} C_VEL
LIN {X 0,Y 727.899,Z 1104.879,A -85,B 0,C 180,E1 34293.544,E2 34293.544} C_VEL
LIN {X 0,Y 727.917,Z 1109.555,A -85,B 0,C 180,E1 34291.653,E2 34291.653} C_VEL
LIN {X 0,Y 727.915,Z 1112.495,A -85,B 0,C 180,E1 34289.921,E2 34289.921} C_VEL
LIN {X 0,Y 727.909,Z 1114.247,A -85,B 0,C 180,E1 34287.874,E2 34287.874} C_VEL
LIN {X 0,Y 727.895,Z 1114.299,A -85,B 0,C 180,E1 34286.219,E2 34286.219} C_VEL
LIN {X 0,Y 727.903,Z 1112.974,A -85,B 0,C 180,E1 34284.324,E2 34284.324} C_VEL
LIN {X 0,Y 727.91,Z 1109.887,A -85,B 0,C 180,E1 34282.422,E2 34282.422} C_VEL
LIN {X 0,Y 727.892,Z 1105.933,A -85,B 0,C 180,E1 34280.751,E2 34280.751} C_VEL
LIN {X 0,Y 727.934,Z 1099.42,A -85,B 0,C 180,E1 34278.741,E2 34278.741} C_VEL
LIN {X 0,Y 727.936,Z 1092.866,A -85,B 0,C 180,E1 34277.143,E2 34277.143} C_VEL
LIN {X 0,Y 728.022,Z 1084.164,A -85,B 0,C 180,E1 34275.362,E2 34275.362} C_VEL
LIN {X 0,Y 728.095,Z 1073.517,A -85,B 0,C 180,E1 34273.567,E2 34273.567} C_VEL
LIN {X 0,Y 728.196,Z 1062.272,A -85,B 0,C 180,E1 34271.921,E2 34271.921} C_VEL
LIN {X 0,Y 728.354,Z 1048.455,A -85,B 0,C 180,E1 34270.179,E2 34270.179} C_VEL
LIN {X 0,Y 728.52,Z 1034.844,A -85,B 0,C 180,E1 34268.672,E2 34268.672} C_VEL
LIN {X 0,Y 728.775,Z 1017.821,A -85,B 0,C 180,E1 34267.018,E2 34267.018} C_VEL
LIN {X 0,Y 729.037,Z 1001.302,A -85,B 0,C 180,E1 34265.602,E2 34265.602} C_VEL
LIN {X 0,Y 729.339,Z 982.036,A -85,B 0,C 180,E1 34264.153,E2 34264.153} C_VEL
LIN {X 0,Y 729.693,Z 963.376,A -85,B 0,C 180,E1 34262.915,E2 34262.915} C_VEL
LIN {X 0,Y 730.038,Z 941.755,A -85,B 0,C 180,E1 34261.668,E2 34261.668} C_VEL
LIN {X 0,Y 730.405,Z 921.575,A -85,B 0,C 180,E1 34260.654,E2 34260.654} C_VEL
LIN {X 0,Y 730.764,Z 898.79,A -85,B 0,C 180,E1 34259.675,E2 34259.675} C_VEL
LIN {X 0,Y 731.025,Z 877.894,A -85,B 0,C 180,E1 34258.913,E2 34258.913} C_VEL
LIN {X 0,Y 731.412,Z 852.57,A -85,B 0,C 180,E1 34258.159,E2 34258.159} C_VEL
LIN {X 0,Y 731.611,Z 831.415,A -85,B 0,C 180,E1 34257.66,E2 34257.66} C_VEL
LIN {X 0,Y 731.876,Z 807.241,A -85,B 0,C 180,E1 34257.225,E2 34257.225} C_VEL
LIN {X 0,Y 732.01,Z 764.198,A -85,B 0,C 180,E1 34256.721,E2 34256.721} C_VEL
LIN {X 0,Y 732.798,Z 517.119,A -85,B 0,C 180,E1 34253.972,E2 34253.972} C_VEL
LIN {X 0,Y 732.917,Z 420.355,A -85,B 0,C 180,E1 34252.864,E2 34252.864} C_VEL
LIN {X 0,Y 731.156,Z 413.59,A -85,B 0,C 180,E1 34252.677,E2 34252.677} C_VEL
LIN {X 0,Y 730.874,Z 409.943,A -85,B 0,C 180,E1 34252.399,E2 34252.399} C_VEL
LIN {X 0,Y 728.103,Z 401.668,A -85,B 0,C 180,E1 34251.581,E2 34251.581} C_VEL
LIN {X 0,Y 728.074,Z 401.537,A -85,B 0,C 180,E1 34248.551,E2 34248.551} C_VEL
LIN {X 0,Y 728.053,Z 401.536,A -85,B 0,C 180,E1 34246.088,E2 34246.088} C_VEL
LIN {X 0,Y 728.067,Z 401.535,A -85,B 0,C 180,E1 34243.748,E2 34243.748} C_VEL
LIN {X 0,Y 728.153,Z 401.523,A -85,B 0,C 180,E1 34240.921,E2 34240.921} C_VEL
LIN {X 0,Y 728.072,Z 401.531,A -85,B 0,C 180,E1 34238.171,E2 34238.171} C_VEL
LIN {X 0,Y 728.07,Z 401.517,A -85,B 0,C 180,E1 34235.806,E2 34235.806} C_VEL
LIN {X 0,Y 728.12,Z 401.532,A -85,B 0,C 180,E1 34233.225,E2 34233.225} C_VEL
LIN {X 0,Y 728.099,Z 401.516,A -85,B 0,C 180,E1 34230.254,E2 34230.254} C_VEL
LIN {X 0,Y 728.082,Z 401.526,A -85,B 0,C 180,E1 34227.746,E2 34227.746} C_VEL
LIN {X 0,Y 728.131,Z 401.533,A -85,B 0,C 180,E1 34225.108,E2 34225.108} C_VEL
LIN {X 0,Y 728.108,Z 401.527,A -85,B 0,C 180,E1 34222.103,E2 34222.103} C_VEL
LIN {X 0,Y 728.097,Z 401.527,A -85,B 0,C 180,E1 34219.494,E2 34219.494} C_VEL
LIN {X 0,Y 728.158,Z 401.525,A -85,B 0,C 180,E1 34216.678,E2 34216.678} C_VEL
LIN {X 0,Y 728.108,Z 401.527,A -85,B 0,C 180,E1 34213.825,E2 34213.825} C_VEL
LIN {X 0,Y 728.127,Z 401.529,A -85,B 0,C 180,E1 34211.084,E2 34211.084} C_VEL
LIN {X 0,Y 728.135,Z 401.522,A -85,B 0,C 180,E1 34207.972,E2 34207.972} C_VEL
LIN {X 0,Y 728.118,Z 401.528,A -85,B 0,C 180,E1 34205.2,E2 34205.2} C_VEL
LIN {X 0,Y 728.152,Z 401.52,A -85,B 0,C 180,E1 34202.282,E2 34202.282} C_VEL
LIN {X 0,Y 728.12,Z 401.526,A -85,B 0,C 180,E1 34199.449,E2 34199.449} C_VEL
LIN {X 0,Y 728.157,Z 401.529,A -85,B 0,C 180,E1 34196.615,E2 34196.615} C_VEL
LIN {X 0,Y 728.138,Z 401.521,A -85,B 0,C 180,E1 34193.614,E2 34193.614} C_VEL
LIN {X 0,Y 728.155,Z 401.532,A -85,B 0,C 180,E1 34190.675,E2 34190.675} C_VEL
LIN {X 0,Y 728.153,Z 401.517,A -85,B 0,C 180,E1 34187.63,E2 34187.63} C_VEL
LIN {X 0,Y 728.159,Z 401.529,A -85,B 0,C 180,E1 34184.55,E2 34184.55} C_VEL
LIN {X 0,Y 728.154,Z 401.521,A -85,B 0,C 180,E1 34181.506,E2 34181.506} C_VEL
LIN {X 0,Y 728.156,Z 401.526,A -85,B 0,C 180,E1 34178.491,E2 34178.491} C_VEL
LIN {X 0,Y 728.159,Z 401.521,A -85,B 0,C 180,E1 34175.413,E2 34175.413} C_VEL
LIN {X 0,Y 728.145,Z 401.531,A -85,B 0,C 180,E1 34172.34,E2 34172.34} C_VEL
LIN {X 0,Y 728.157,Z 401.519,A -85,B 0,C 180,E1 34169.373,E2 34169.373} C_VEL
LIN {X 0,Y 728.145,Z 401.531,A -85,B 0,C 180,E1 34166.305,E2 34166.305} C_VEL
LIN {X 0,Y 728.137,Z 401.523,A -85,B 0,C 180,E1 34163.418,E2 34163.418} C_VEL
LIN {X 0,Y 728.153,Z 401.529,A -85,B 0,C 180,E1 34160.386,E2 34160.386} C_VEL
LIN {X 0,Y 728.115,Z 401.523,A -85,B 0,C 180,E1 34157.602,E2 34157.602} C_VEL
LIN {X 0,Y 728.156,Z 401.527,A -85,B 0,C 180,E1 34154.77,E2 34154.77} C_VEL
LIN {X 0,Y 728.11,Z 401.532,A -85,B 0,C 180,E1 34151.868,E2 34151.868} C_VEL
LIN {X 0,Y 728.121,Z 401.529,A -85,B 0,C 180,E1 34149.175,E2 34149.175} C_VEL
LIN {X 0,Y 728.165,Z 401.801,A -85,B 0,C 180,E1 34148.065,E2 34148.065} C_VEL
LIN {X 0,Y 731.902,Z 412.161,A -85,B 0,C 180,E1 34147.076,E2 34147.076} C_VEL
LIN {X 0,Y 731.331,Z 447.924,A -85,B 0,C 180,E1 34144.607,E2 34144.607} C_VEL
LIN {X 0,Y 731.425,Z 453.594,A -85,B 0,C 180,E1 34144.251,E2 34144.251} C_VEL
LIN {X 0,Y 733.116,Z 461.184,A -85,B 0,C 180,E1 34144.071,E2 34144.071} C_VEL
LIN {X 0,Y 732.281,Z 713.507,A -85,B 0,C 180,E1 34141.235,E2 34141.235} C_VEL
LIN {X 0,Y 731.896,Z 842.73,A -85,B 0,C 180,E1 34139.788,E2 34139.788} C_VEL
LIN {X 0,Y 731.63,Z 868.109,A -85,B 0,C 180,E1 34139.365,E2 34139.365} C_VEL
LIN {X 0,Y 731.416,Z 889.68,A -85,B 0,C 180,E1 34138.87,E2 34138.87} C_VEL
LIN {X 0,Y 731.15,Z 913.285,A -85,B 0,C 180,E1 34138.196,E2 34138.196} C_VEL
LIN {X 0,Y 730.784,Z 936.272,A -85,B 0,C 180,E1 34137.378,E2 34137.378} C_VEL
LIN {X 0,Y 730.481,Z 958.075,A -85,B 0,C 180,E1 34136.465,E2 34136.465} C_VEL
LIN {X 0,Y 730.06,Z 979.943,A -85,B 0,C 180,E1 34135.384,E2 34135.384} C_VEL
LIN {X 0,Y 729.749,Z 1000.341,A -85,B 0,C 180,E1 34134.228,E2 34134.228} C_VEL
LIN {X 0,Y 729.366,Z 1020.441,A -85,B 0,C 180,E1 34132.913,E2 34132.913} C_VEL
LIN {X 0,Y 729.084,Z 1039.25,A -85,B 0,C 180,E1 34131.522,E2 34131.522} C_VEL
LIN {X 0,Y 728.776,Z 1056.46,A -85,B 0,C 180,E1 34130.06,E2 34130.06} C_VEL
LIN {X 0,Y 728.567,Z 1072.961,A -85,B 0,C 180,E1 34128.483,E2 34128.483} C_VEL
LIN {X 0,Y 728.355,Z 1087.454,A -85,B 0,C 180,E1 34126.893,E2 34126.893} C_VEL
LIN {X 0,Y 728.207,Z 1101.057,A -85,B 0,C 180,E1 34125.204,E2 34125.204} C_VEL
LIN {X 0,Y 728.086,Z 1112.793,A -85,B 0,C 180,E1 34123.501,E2 34123.501} C_VEL
LIN {X 0,Y 728.02,Z 1122.95,A -85,B 0,C 180,E1 34121.809,E2 34121.809} C_VEL
LIN {X 0,Y 727.95,Z 1132.181,A -85,B 0,C 180,E1 34119.966,E2 34119.966} C_VEL
LIN {X 0,Y 727.932,Z 1138.815,A -85,B 0,C 180,E1 34118.372,E2 34118.372} C_VEL
LIN {X 0,Y 727.912,Z 1145.245,A -85,B 0,C 180,E1 34116.467,E2 34116.467} C_VEL
LIN {X 0,Y 727.917,Z 1149.813,A -85,B 0,C 180,E1 34114.57,E2 34114.57} C_VEL
LIN {X 0,Y 727.882,Z 1152.684,A -85,B 0,C 180,E1 34112.835,E2 34112.835} C_VEL
LIN {X 0,Y 727.89,Z 1154.262,A -85,B 0,C 180,E1 34110.866,E2 34110.866} C_VEL
LIN {X 0,Y 727.883,Z 1154.306,A -85,B 0,C 180,E1 34109.292,E2 34109.292} C_VEL
LIN {X 0,Y 727.89,Z 1153.017,A -85,B 0,C 180,E1 34107.402,E2 34107.402} C_VEL
LIN {X 0,Y 727.916,Z 1149.971,A -85,B 0,C 180,E1 34105.509,E2 34105.509} C_VEL
LIN {X 0,Y 727.92,Z 1145.864,A -85,B 0,C 180,E1 34103.77,E2 34103.77} C_VEL
LIN {X 0,Y 727.942,Z 1139.422,A -85,B 0,C 180,E1 34101.787,E2 34101.787} C_VEL
LIN {X 0,Y 727.944,Z 1132.891,A -85,B 0,C 180,E1 34100.193,E2 34100.193} C_VEL
LIN {X 0,Y 728.023,Z 1124.295,A -85,B 0,C 180,E1 34098.433,E2 34098.433} C_VEL
LIN {X 0,Y 728.073,Z 1113.834,A -85,B 0,C 180,E1 34096.66,E2 34096.66} C_VEL
LIN {X 0,Y 728.18,Z 1103.376,A -85,B 0,C 180,E1 34095.121,E2 34095.121} C_VEL
LIN {X 0,Y 728.356,Z 1088.632,A -85,B 0,C 180,E1 34093.244,E2 34093.244} C_VEL
LIN {X 0,Y 728.507,Z 1075.291,A -85,B 0,C 180,E1 34091.764,E2 34091.764} C_VEL
LIN {X 0,Y 728.757,Z 1058.318,A -85,B 0,C 180,E1 34090.107,E2 34090.107} C_VEL
LIN {X 0,Y 729.027,Z 1041.791,A -85,B 0,C 180,E1 34088.687,E2 34088.687} C_VEL
LIN {X 0,Y 729.342,Z 1022.252,A -85,B 0,C 180,E1 34087.214,E2 34087.214} C_VEL
LIN {X 0,Y 729.684,Z 1003.76,A -85,B 0,C 180,E1 34085.985,E2 34085.985} C_VEL
LIN {X 0,Y 730.032,Z 982.347,A -85,B 0,C 180,E1 34084.745,E2 34084.745} C_VEL
LIN {X 0,Y 730.389,Z 962.155,A -85,B 0,C 180,E1 34083.726,E2 34083.726} C_VEL
LIN {X 0,Y 730.764,Z 938.712,A -85,B 0,C 180,E1 34082.718,E2 34082.718} C_VEL
LIN {X 0,Y 731.018,Z 918.423,A -85,B 0,C 180,E1 34081.976,E2 34081.976} C_VEL
LIN {X 0,Y 731.401,Z 892.947,A -85,B 0,C 180,E1 34081.214,E2 34081.214} C_VEL
LIN {X 0,Y 731.604,Z 871.754,A -85,B 0,C 180,E1 34080.712,E2 34080.712} C_VEL
LIN {X 0,Y 731.874,Z 847.924,A -85,B 0,C 180,E1 34080.28,E2 34080.28} C_VEL
LIN {X 0,Y 732.008,Z 806.775,A -85,B 0,C 180,E1 34079.795,E2 34079.795} C_VEL
LIN {X 0,Y 732.656,Z 578.503,A -85,B 0,C 180,E1 34077.254,E2 34077.254} C_VEL
LIN {X 0,Y 732.949,Z 459.587,A -85,B 0,C 180,E1 34075.902,E2 34075.902} C_VEL
LIN {X 0,Y 731.304,Z 452.723,A -85,B 0,C 180,E1 34075.714,E2 34075.714} C_VEL
LIN {X 0,Y 731.838,Z 416.705,A -85,B 0,C 180,E1 34073.242,E2 34073.242} C_VEL
LIN {X 0,Y 731.707,Z 411.18,A -85,B 0,C 180,E1 34072.843,E2 34072.843} C_VEL
LIN {X 0,Y 728.165,Z 401.799,A -85,B 0,C 180,E1 34071.935,E2 34071.935} C_VEL
LIN {X 0,Y 728.109,Z 401.527,A -85,B 0,C 180,E1 34070.11,E2 34070.11} C_VEL
LIN {X 0,Y 728.157,Z 401.527,A -85,B 0,C 180,E1 34067.162,E2 34067.162} C_VEL
LIN {X 0,Y 728.11,Z 401.529,A -85,B 0,C 180,E1 34064.318,E2 34064.318} C_VEL
LIN {X 0,Y 728.159,Z 401.515,A -85,B 0,C 180,E1 34061.548,E2 34061.548} C_VEL
LIN {X 0,Y 728.131,Z 401.525,A -85,B 0,C 180,E1 34058.568,E2 34058.568} C_VEL
LIN {X 0,Y 728.143,Z 401.529,A -85,B 0,C 180,E1 34055.705,E2 34055.705} C_VEL
LIN {X 0,Y 728.153,Z 401.519,A -85,B 0,C 180,E1 34052.661,E2 34052.661} C_VEL
LIN {X 0,Y 728.138,Z 401.531,A -85,B 0,C 180,E1 34049.718,E2 34049.718} C_VEL
LIN {X 0,Y 728.151,Z 401.523,A -85,B 0,C 180,E1 34046.77,E2 34046.77} C_VEL
LIN {X 0,Y 728.132,Z 401.524,A -85,B 0,C 180,E1 34043.855,E2 34043.855} C_VEL
LIN {X 0,Y 728.142,Z 401.527,A -85,B 0,C 180,E1 34041.087,E2 34041.087} C_VEL
LIN {X 0,Y 728.142,Z 401.52,A -85,B 0,C 180,E1 34038.146,E2 34038.146} C_VEL
LIN {X 0,Y 728.148,Z 401.527,A -85,B 0,C 180,E1 34035.206,E2 34035.206} C_VEL
LIN {X 0,Y 728.156,Z 401.52,A -85,B 0,C 180,E1 34032.209,E2 34032.209} C_VEL
LIN {X 0,Y 728.146,Z 401.527,A -85,B 0,C 180,E1 34029.166,E2 34029.166} C_VEL
LIN {X 0,Y 728.158,Z 401.52,A -85,B 0,C 180,E1 34026.149,E2 34026.149} C_VEL
LIN {X 0,Y 728.14,Z 401.528,A -85,B 0,C 180,E1 34023.07,E2 34023.07} C_VEL
LIN {X 0,Y 728.144,Z 401.522,A -85,B 0,C 180,E1 34020.157,E2 34020.157} C_VEL
LIN {X 0,Y 728.145,Z 401.53,A -85,B 0,C 180,E1 34017.088,E2 34017.088} C_VEL
LIN {X 0,Y 728.122,Z 401.524,A -85,B 0,C 180,E1 34014.247,E2 34014.247} C_VEL
LIN {X 0,Y 728.157,Z 401.526,A -85,B 0,C 180,E1 34011.312,E2 34011.312} C_VEL
LIN {X 0,Y 728.107,Z 401.528,A -85,B 0,C 180,E1 34008.514,E2 34008.514} C_VEL
LIN {X 0,Y 728.103,Z 401.523,A -85,B 0,C 180,E1 34006.402,E2 34006.402} C_VEL
LIN {X 0,Y 727.109,Z 401.651,A -85,B 0,C 180,E1 34005.796,E2 34005.796} C_VEL
LIN {X 0,Y 720.705,Z 402.451,A -85,B 0,C 180,E1 34004.098,E2 34004.098} C_VEL
LIN {X 0,Y 720.215,Z 402.513,A -85,B 0,C 180,E1 34003.657,E2 34003.657} C_VEL
LIN {X 0,Y 720.175,Z 402.517,A -85,B 0,C 180,E1 34000.704,E2 34000.704} C_VEL
LIN {X 0,Y 720.16,Z 402.516,A -85,B 0,C 180,E1 33998.044,E2 33998.044} C_VEL
LIN {X 0,Y 720.22,Z 402.515,A -85,B 0,C 180,E1 33995.124,E2 33995.124} C_VEL
LIN {X 0,Y 720.15,Z 402.516,A -85,B 0,C 180,E1 33992.354,E2 33992.354} C_VEL
LIN {X 0,Y 720.158,Z 402.517,A -85,B 0,C 180,E1 33989.827,E2 33989.827} C_VEL
LIN {X 0,Y 720.196,Z 402.52,A -85,B 0,C 180,E1 33986.837,E2 33986.837} C_VEL
LIN {X 0,Y 720.136,Z 402.519,A -85,B 0,C 180,E1 33984.181,E2 33984.181} C_VEL
LIN {X 0,Y 720.142,Z 402.52,A -85,B 0,C 180,E1 33981.738,E2 33981.738} C_VEL
LIN {X 0,Y 720.204,Z 402.505,A -85,B 0,C 180,E1 33978.847,E2 33978.847} C_VEL
LIN {X 0,Y 720.125,Z 402.52,A -85,B 0,C 180,E1 33976.107,E2 33976.107} C_VEL
LIN {X 0,Y 720.123,Z 402.521,A -85,B 0,C 180,E1 33973.747,E2 33973.747} C_VEL
LIN {X 0,Y 720.206,Z 402.505,A -85,B 0,C 180,E1 33970.942,E2 33970.942} C_VEL
LIN {X 0,Y 720.121,Z 402.517,A -85,B 0,C 180,E1 33968.162,E2 33968.162} C_VEL
LIN {X 0,Y 720.11,Z 402.527,A -85,B 0,C 180,E1 33965.816,E2 33965.816} C_VEL
LIN {X 0,Y 720.127,Z 402.531,A -85,B 0,C 180,E1 33963.437,E2 33963.437} C_VEL
LIN {X 0,Y 720.236,Z 402.712,A -85,B 0,C 180,E1 33962.687,E2 33962.687} C_VEL
LIN {X 0,Y 723.984,Z 413.82,A -85,B 0,C 180,E1 33961.611,E2 33961.611} C_VEL
LIN {X 0,Y 726.475,Z 423.699,A -85,B 0,C 180,E1 33961.352,E2 33961.352} C_VEL
LIN {X 0,Y 725.437,Z 674.871,A -85,B 0,C 180,E1 33958.503,E2 33958.503} C_VEL
LIN {X 0,Y 724.932,Z 802.821,A -85,B 0,C 180,E1 33957.058,E2 33957.058} C_VEL
LIN {X 0,Y 724.629,Z 828.122,A -85,B 0,C 180,E1 33956.632,E2 33956.632} C_VEL
LIN {X 0,Y 724.35,Z 849.891,A -85,B 0,C 180,E1 33956.129,E2 33956.129} C_VEL
LIN {X 0,Y 723.994,Z 873.8,A -85,B 0,C 180,E1 33955.437,E2 33955.437} C_VEL
LIN {X 0,Y 723.546,Z 896.447,A -85,B 0,C 180,E1 33954.623,E2 33954.623} C_VEL
LIN {X 0,Y 723.137,Z 919.557,A -85,B 0,C 180,E1 33953.64,E2 33953.64} C_VEL
LIN {X 0,Y 722.632,Z 940.664,A -85,B 0,C 180,E1 33952.58,E2 33952.58} C_VEL
LIN {X 0,Y 722.214,Z 961.935,A -85,B 0,C 180,E1 33951.353,E2 33951.353} C_VEL
LIN {X 0,Y 721.75,Z 981.229,A -85,B 0,C 180,E1 33950.068,E2 33950.068} C_VEL
LIN {X 0,Y 721.376,Z 1000.279,A -85,B 0,C 180,E1 33948.632,E2 33948.632} C_VEL
LIN {X 0,Y 721.016,Z 1017.114,A -85,B 0,C 180,E1 33947.181,E2 33947.181} C_VEL
LIN {X 0,Y 720.727,Z 1034.033,A -85,B 0,C 180,E1 33945.531,E2 33945.531} C_VEL
LIN {X 0,Y 720.472,Z 1047.997,A -85,B 0,C 180,E1 33943.974,E2 33943.974} C_VEL
LIN {X 0,Y 720.285,Z 1062.108,A -85,B 0,C 180,E1 33942.181,E2 33942.181} C_VEL
LIN {X 0,Y 720.15,Z 1073.608,A -85,B 0,C 180,E1 33940.48,E2 33940.48} C_VEL
LIN {X 0,Y 720.046,Z 1084.495,A -85,B 0,C 180,E1 33938.613,E2 33938.613} C_VEL
LIN {X 0,Y 719.951,Z 1092.943,A -85,B 0,C 180,E1 33936.86,E2 33936.86} C_VEL
LIN {X 0,Y 719.938,Z 1099.484,A -85,B 0,C 180,E1 33935.243,E2 33935.243} C_VEL
LIN {X 0,Y 719.893,Z 1105.838,A -85,B 0,C 180,E1 33933.265,E2 33933.265} C_VEL
LIN {X 0,Y 719.915,Z 1109.781,A -85,B 0,C 180,E1 33931.592,E2 33931.592} C_VEL
LIN {X 0,Y 719.908,Z 1112.768,A -85,B 0,C 180,E1 33929.761,E2 33929.761} C_VEL
LIN {X 0,Y 719.902,Z 1114.278,A -85,B 0,C 180,E1 33927.771,E2 33927.771} C_VEL
LIN {X 0,Y 719.9,Z 1114.267,A -85,B 0,C 180,E1 33926.098,E2 33926.098} C_VEL
LIN {X 0,Y 719.91,Z 1112.588,A -85,B 0,C 180,E1 33924.021,E2 33924.021} C_VEL
LIN {X 0,Y 719.917,Z 1109.66,A -85,B 0,C 180,E1 33922.257,E2 33922.257} C_VEL
LIN {X 0,Y 719.904,Z 1104.982,A -85,B 0,C 180,E1 33920.325,E2 33920.325} C_VEL
LIN {X 0,Y 719.929,Z 1099.023,A -85,B 0,C 180,E1 33918.544,E2 33918.544} C_VEL
LIN {X 0,Y 719.958,Z 1092.353,A -85,B 0,C 180,E1 33916.916,E2 33916.916} C_VEL
LIN {X 0,Y 720.039,Z 1083.049,A -85,B 0,C 180,E1 33915.031,E2 33915.031} C_VEL
LIN {X 0,Y 720.155,Z 1073.041,A -85,B 0,C 180,E1 33913.341,E2 33913.341} C_VEL
LIN {X 0,Y 720.312,Z 1060.833,A -85,B 0,C 180,E1 33911.549,E2 33911.549} C_VEL
LIN {X 0,Y 720.475,Z 1047.421,A -85,B 0,C 180,E1 33909.868,E2 33909.868} C_VEL
LIN {X 0,Y 720.754,Z 1032.917,A -85,B 0,C 180,E1 33908.259,E2 33908.259} C_VEL
LIN {X 0,Y 721.021,Z 1017,A -85,B 0,C 180,E1 33906.72,E2 33906.72} C_VEL
LIN {X 0,Y 721.383,Z 999.996,A -85,B 0,C 180,E1 33905.254,E2 33905.254} C_VEL
LIN {X 0,Y 721.76,Z 980.879,A -85,B 0,C 180,E1 33903.817,E2 33903.817} C_VEL
LIN {X 0,Y 722.235,Z 961.289,A -85,B 0,C 180,E1 33902.515,E2 33902.515} C_VEL
LIN {X 0,Y 722.648,Z 940.218,A -85,B 0,C 180,E1 33901.306,E2 33901.306} C_VEL
LIN {X 0,Y 723.17,Z 917.924,A -85,B 0,C 180,E1 33900.194,E2 33900.194} C_VEL
LIN {X 0,Y 723.561,Z 895.497,A -85,B 0,C 180,E1 33899.249,E2 33899.249} C_VEL
LIN {X 0,Y 724.037,Z 872.057,A -85,B 0,C 180,E1 33898.416,E2 33898.416} C_VEL
LIN {X 0,Y 724.364,Z 848.383,A -85,B 0,C 180,E1 33897.742,E2 33897.742} C_VEL
LIN {X 0,Y 724.729,Z 824.5,A -85,B 0,C 180,E1 33897.204,E2 33897.204} C_VEL
LIN {X 0,Y 724.939,Z 800.46,A -85,B 0,C 180,E1 33896.821,E2 33896.821} C_VEL
LIN {X 0,Y 725.992,Z 536.441,A -85,B 0,C 180,E1 33893.847,E2 33893.847} C_VEL
LIN {X 0,Y 726.286,Z 422.233,A -85,B 0,C 180,E1 33892.531,E2 33892.531} C_VEL
LIN {X 0,Y 723.893,Z 413.636,A -85,B 0,C 180,E1 33892.288,E2 33892.288} C_VEL
LIN {X 0,Y 720.225,Z 402.673,A -85,B 0,C 180,E1 33891.216,E2 33891.216} C_VEL
LIN {X 0,Y 720.119,Z 402.527,A -85,B 0,C 180,E1 33888.333,E2 33888.333} C_VEL
LIN {X 0,Y 720.117,Z 402.526,A -85,B 0,C 180,E1 33885.921,E2 33885.921} C_VEL
LIN {X 0,Y 720.177,Z 402.525,A -85,B 0,C 180,E1 33883.304,E2 33883.304} C_VEL
LIN {X 0,Y 720.139,Z 402.519,A -85,B 0,C 180,E1 33880.318,E2 33880.318} C_VEL
LIN {X 0,Y 720.129,Z 402.52,A -85,B 0,C 180,E1 33877.939,E2 33877.939} C_VEL
LIN {X 0,Y 720.15,Z 402.504,A -85,B 0,C 180,E1 33875.477,E2 33875.477} C_VEL
LIN {X 0,Y 720.172,Z 402.517,A -85,B 0,C 180,E1 33872.407,E2 33872.407} C_VEL
LIN {X 0,Y 720.14,Z 402.504,A -85,B 0,C 180,E1 33869.898,E2 33869.898} C_VEL
LIN {X 0,Y 720.165,Z 402.516,A -85,B 0,C 180,E1 33867.359,E2 33867.359} C_VEL
LIN {X 0,Y 720.182,Z 402.512,A -85,B 0,C 180,E1 33864.265,E2 33864.265} C_VEL
LIN {X 0,Y 720.152,Z 402.519,A -85,B 0,C 180,E1 33861.674,E2 33861.674} C_VEL
LIN {X 0,Y 720.207,Z 402.519,A -85,B 0,C 180,E1 33858.958,E2 33858.958} C_VEL
LIN {X 0,Y 720.173,Z 402.51,A -85,B 0,C 180,E1 33855.956,E2 33855.956} C_VEL
LIN {X 0,Y 720.175,Z 402.52,A -85,B 0,C 180,E1 33853.243,E2 33853.243} C_VEL
LIN {X 0,Y 720.218,Z 402.512,A -85,B 0,C 180,E1 33850.236,E2 33850.236} C_VEL
LIN {X 0,Y 720.17,Z 402.516,A -85,B 0,C 180,E1 33847.419,E2 33847.419} C_VEL
LIN {X 0,Y 720.217,Z 402.518,A -85,B 0,C 180,E1 33844.573,E2 33844.573} C_VEL
LIN {X 0,Y 720.186,Z 402.508,A -85,B 0,C 180,E1 33841.671,E2 33841.671} C_VEL
LIN {X 0,Y 720.212,Z 402.521,A -85,B 0,C 180,E1 33838.807,E2 33838.807} C_VEL
LIN {X 0,Y 720.202,Z 402.51,A -85,B 0,C 180,E1 33835.7,E2 33835.7} C_VEL
LIN {X 0,Y 720.216,Z 402.517,A -85,B 0,C 180,E1 33832.742,E2 33832.742} C_VEL
LIN {X 0,Y 720.214,Z 402.51,A -85,B 0,C 180,E1 33829.683,E2 33829.683} C_VEL
LIN {X 0,Y 720.218,Z 402.517,A -85,B 0,C 180,E1 33826.676,E2 33826.676} C_VEL
LIN {X 0,Y 720.216,Z 402.506,A -85,B 0,C 180,E1 33823.548,E2 33823.548} C_VEL
LIN {X 0,Y 720.215,Z 402.52,A -85,B 0,C 180,E1 33820.506,E2 33820.506} C_VEL
LIN {X 0,Y 720.222,Z 402.505,A -85,B 0,C 180,E1 33817.47,E2 33817.47} C_VEL
LIN {X 0,Y 720.21,Z 402.516,A -85,B 0,C 180,E1 33814.42,E2 33814.42} C_VEL
LIN {X 0,Y 720.219,Z 402.51,A -85,B 0,C 180,E1 33811.382,E2 33811.382} C_VEL
LIN {X 0,Y 720.206,Z 402.517,A -85,B 0,C 180,E1 33808.327,E2 33808.327} C_VEL
LIN {X 0,Y 720.205,Z 402.51,A -85,B 0,C 180,E1 33805.401,E2 33805.401} C_VEL
LIN {X 0,Y 720.209,Z 402.52,A -85,B 0,C 180,E1 33802.312,E2 33802.312} C_VEL
LIN {X 0,Y 720.189,Z 402.515,A -85,B 0,C 180,E1 33799.415,E2 33799.415} C_VEL
LIN {X 0,Y 720.214,Z 402.521,A -85,B 0,C 180,E1 33796.37,E2 33796.37} C_VEL
LIN {X 0,Y 720.171,Z 402.519,A -85,B 0,C 180,E1 33793.524,E2 33793.524} C_VEL
LIN {X 0,Y 720.219,Z 402.521,A -85,B 0,C 180,E1 33790.626,E2 33790.626} C_VEL
LIN {X 0,Y 720.251,Z 402.739,A -85,B 0,C 180,E1 33788.496,E2 33788.496} C_VEL
LIN {X 0,Y 724.916,Z 415.381,A -85,B 0,C 180,E1 33787.262,E2 33787.262} C_VEL
LIN {X 0,Y 724.218,Z 451.232,A -85,B 0,C 180,E1 33784.765,E2 33784.765} C_VEL
LIN {X 0,Y 724.415,Z 453.935,A -85,B 0,C 180,E1 33784.623,E2 33784.623} C_VEL
LIN {X 0,Y 726.475,Z 462.837,A -85,B 0,C 180,E1 33784.407,E2 33784.407} C_VEL
LIN {X 0,Y 725.432,Z 714.525,A -85,B 0,C 180,E1 33781.552,E2 33781.552} C_VEL
LIN {X 0,Y 724.941,Z 842.837,A -85,B 0,C 180,E1 33780.102,E2 33780.102} C_VEL
LIN {X 0,Y 724.618,Z 868.368,A -85,B 0,C 180,E1 33779.672,E2 33779.672} C_VEL
LIN {X 0,Y 724.342,Z 890.115,A -85,B 0,C 180,E1 33779.168,E2 33779.168} C_VEL
LIN {X 0,Y 724.014,Z 913.281,A -85,B 0,C 180,E1 33778.499,E2 33778.499} C_VEL
LIN {X 0,Y 723.568,Z 935.358,A -85,B 0,C 180,E1 33777.711,E2 33777.711} C_VEL
LIN {X 0,Y 723.176,Z 957.231,A -85,B 0,C 180,E1 33776.791,E2 33776.791} C_VEL
LIN {X 0,Y 722.68,Z 979.144,A -85,B 0,C 180,E1 33775.706,E2 33775.706} C_VEL
LIN {X 0,Y 722.248,Z 999.617,A -85,B 0,C 180,E1 33774.54,E2 33774.54} C_VEL
LIN {X 0,Y 721.8,Z 1019.839,A -85,B 0,C 180,E1 33773.211,E2 33773.211} C_VEL
LIN {X 0,Y 721.413,Z 1038.708,A -85,B 0,C 180,E1 33771.805,E2 33771.805} C_VEL
LIN {X 0,Y 721.03,Z 1056.46,A -85,B 0,C 180,E1 33770.285,E2 33770.285} C_VEL
LIN {X 0,Y 720.756,Z 1072.963,A -85,B 0,C 180,E1 33768.691,E2 33768.691} C_VEL
LIN {X 0,Y 720.478,Z 1087.219,A -85,B 0,C 180,E1 33767.111,E2 33767.111} C_VEL
LIN {X 0,Y 720.295,Z 1101.059,A -85,B 0,C 180,E1 33765.375,E2 33765.375} C_VEL
LIN {X 0,Y 720.142,Z 1113.081,A -85,B 0,C 180,E1 33763.608,E2 33763.608} C_VEL
LIN {X 0,Y 720.049,Z 1123.867,A -85,B 0,C 180,E1 33761.779,E2 33761.779} C_VEL
LIN {X 0,Y 719.96,Z 1132.892,A -85,B 0,C 180,E1 33759.917,E2 33759.917} C_VEL
LIN {X 0,Y 719.944,Z 1139.423,A -85,B 0,C 180,E1 33758.305,E2 33758.305} C_VEL
LIN {X 0,Y 719.92,Z 1146.07,A -85,B 0,C 180,E1 33756.219,E2 33756.219} C_VEL
LIN {X 0,Y 719.917,Z 1149.972,A -85,B 0,C 180,E1 33754.541,E2 33754.541} C_VEL
LIN {X 0,Y 719.888,Z 1153.017,A -85,B 0,C 180,E1 33752.627,E2 33752.627} C_VEL
LIN {X 0,Y 719.883,Z 1154.306,A -85,B 0,C 180,E1 33750.716,E2 33750.716} C_VEL
LIN {X 0,Y 719.896,Z 1154.24,A -85,B 0,C 180,E1 33749.045,E2 33749.045} C_VEL
LIN {X 0,Y 719.882,Z 1152.559,A -85,B 0,C 180,E1 33747.045,E2 33747.045} C_VEL
LIN {X 0,Y 719.916,Z 1149.813,A -85,B 0,C 180,E1 33745.379,E2 33745.379} C_VEL
LIN {X 0,Y 719.916,Z 1145.245,A -85,B 0,C 180,E1 33743.46,E2 33743.46} C_VEL
LIN {X 0,Y 719.934,Z 1138.815,A -85,B 0,C 180,E1 33741.534,E2 33741.534} C_VEL
LIN {X 0,Y 719.973,Z 1132.181,A -85,B 0,C 180,E1 33739.922,E2 33739.922} C_VEL
LIN {X 0,Y 720.055,Z 1122.031,A -85,B 0,C 180,E1 33737.896,E2 33737.896} C_VEL
LIN {X 0,Y 720.156,Z 1112.277,A -85,B 0,C 180,E1 33736.265,E2 33736.265} C_VEL
LIN {X 0,Y 720.315,Z 1099.681,A -85,B 0,C 180,E1 33734.444,E2 33734.444} C_VEL
LIN {X 0,Y 720.49,Z 1086.512,A -85,B 0,C 180,E1 33732.806,E2 33732.806} C_VEL
LIN {X 0,Y 720.782,Z 1071.334,A -85,B 0,C 180,E1 33731.142,E2 33731.142} C_VEL
LIN {X 0,Y 721.057,Z 1055.43,A -85,B 0,C 180,E1 33729.622,E2 33729.622} C_VEL
LIN {X 0,Y 721.426,Z 1037.603,A -85,B 0,C 180,E1 33728.11,E2 33728.11} C_VEL
LIN {X 0,Y 721.817,Z 1019.235,A -85,B 0,C 180,E1 33726.747,E2 33726.747} C_VEL
LIN {X 0,Y 722.275,Z 997.433,A -85,B 0,C 180,E1 33725.33,E2 33725.33} C_VEL
LIN {X 0,Y 722.725,Z 977.524,A -85,B 0,C 180,E1 33724.208,E2 33724.208} C_VEL
LIN {X 0,Y 723.206,Z 954.252,A -85,B 0,C 180,E1 33723.077,E2 33723.077} C_VEL
LIN {X 0,Y 723.625,Z 933.106,A -85,B 0,C 180,E1 33722.202,E2 33722.202} C_VEL
LIN {X 0,Y 724.069,Z 908.958,A -85,B 0,C 180,E1 33721.368,E2 33721.368} C_VEL
LIN {X 0,Y 724.364,Z 887.095,A -85,B 0,C 180,E1 33720.754,E2 33720.754} C_VEL
LIN {X 0,Y 724.745,Z 862.437,A -85,B 0,C 180,E1 33720.212,E2 33720.212} C_VEL
LIN {X 0,Y 724.951,Z 839.812,A -85,B 0,C 180,E1 33719.858,E2 33719.858} C_VEL
LIN {X 0,Y 725.894,Z 587.615,A -85,B 0,C 180,E1 33717.016,E2 33717.016} C_VEL
LIN {X 0,Y 726.28,Z 461.253,A -85,B 0,C 180,E1 33715.564,E2 33715.564} C_VEL
LIN {X 0,Y 724.226,Z 452.729,A -85,B 0,C 180,E1 33715.332,E2 33715.332} C_VEL
LIN {X 0,Y 724.884,Z 417.276,A -85,B 0,C 180,E1 33712.872,E2 33712.872} C_VEL
LIN {X 0,Y 724.753,Z 414.847,A -85,B 0,C 180,E1 33712.689,E2 33712.689} C_VEL
LIN {X 0,Y 720.265,Z 402.83,A -85,B 0,C 180,E1 33711.52,E2 33711.52} C_VEL
LIN {X 0,Y 720.167,Z 402.515,A -85,B 0,C 180,E1 33710.616,E2 33710.616} C_VEL
LIN {X 0,Y 720.19,Z 402.518,A -85,B 0,C 180,E1 33707.888,E2 33707.888} C_VEL
LIN {X 0,Y 720.199,Z 402.514,A -85,B 0,C 180,E1 33704.81,E2 33704.81} C_VEL
LIN {X 0,Y 720.179,Z 402.507,A -85,B 0,C 180,E1 33702.006,E2 33702.006} C_VEL
LIN {X 0,Y 720.215,Z 402.515,A -85,B 0,C 180,E1 33699.072,E2 33699.072} C_VEL
LIN {X 0,Y 720.179,Z 402.512,A -85,B 0,C 180,E1 33696.229,E2 33696.229} C_VEL
LIN {X 0,Y 720.214,Z 402.515,A -85,B 0,C 180,E1 33693.352,E2 33693.352} C_VEL
LIN {X 0,Y 720.194,Z 402.513,A -85,B 0,C 180,E1 33690.356,E2 33690.356} C_VEL
LIN {X 0,Y 720.217,Z 402.519,A -85,B 0,C 180,E1 33687.447,E2 33687.447} C_VEL
LIN {X 0,Y 720.209,Z 402.506,A -85,B 0,C 180,E1 33684.39,E2 33684.39} C_VEL
LIN {X 0,Y 720.221,Z 402.522,A -85,B 0,C 180,E1 33681.415,E2 33681.415} C_VEL
LIN {X 0,Y 720.216,Z 402.507,A -85,B 0,C 180,E1 33678.37,E2 33678.37} C_VEL
LIN {X 0,Y 720.218,Z 402.516,A -85,B 0,C 180,E1 33675.295,E2 33675.295} C_VEL
LIN {X 0,Y 720.218,Z 402.509,A -85,B 0,C 180,E1 33672.21,E2 33672.21} C_VEL
LIN {X 0,Y 720.209,Z 402.514,A -85,B 0,C 180,E1 33669.187,E2 33669.187} C_VEL
LIN {X 0,Y 720.22,Z 402.509,A -85,B 0,C 180,E1 33666.137,E2 33666.137} C_VEL
LIN {X 0,Y 720.204,Z 402.516,A -85,B 0,C 180,E1 33663.104,E2 33663.104} C_VEL
LIN {X 0,Y 720.205,Z 402.511,A -85,B 0,C 180,E1 33660.159,E2 33660.159} C_VEL
LIN {X 0,Y 720.204,Z 402.518,A -85,B 0,C 180,E1 33657.055,E2 33657.055} C_VEL
LIN {X 0,Y 720.188,Z 402.513,A -85,B 0,C 180,E1 33654.183,E2 33654.183} C_VEL
LIN {X 0,Y 720.213,Z 402.517,A -85,B 0,C 180,E1 33651.135,E2 33651.135} C_VEL
LIN {X 0,Y 720.17,Z 402.515,A -85,B 0,C 180,E1 33648.305,E2 33648.305} C_VEL
LIN {X 0,Y 720.218,Z 402.51,A -85,B 0,C 180,E1 33645.446,E2 33645.446} C_VEL
LIN {X 0,Y 720.215,Z 402.513,A -85,B 0,C 180,E1 33643.657,E2 33643.657} C_VEL
LIN {X 0,Y 719.283,Z 402.636,A -85,B 0,C 180,E1 33643.044,E2 33643.044} C_VEL
LIN {X 0,Y 712.732,Z 403.448,A -85,B 0,C 180,E1 33641.284,E2 33641.284} C_VEL
LIN {X 0,Y 712.253,Z 403.506,A -85,B 0,C 180,E1 33640.882,E2 33640.882} C_VEL
LIN {X 0,Y 712.217,Z 403.506,A -85,B 0,C 180,E1 33638.159,E2 33638.159} C_VEL
LIN {X 0,Y 712.283,Z 403.497,A -85,B 0,C 180,E1 33635.359,E2 33635.359} C_VEL
LIN {X 0,Y 712.218,Z 403.506,A -85,B 0,C 180,E1 33632.491,E2 33632.491} C_VEL
LIN {X 0,Y 712.212,Z 403.506,A -85,B 0,C 180,E1 33629.92,E2 33629.92} C_VEL
LIN {X 0,Y 712.278,Z 403.505,A -85,B 0,C 180,E1 33626.998,E2 33626.998} C_VEL
LIN {X 0,Y 712.2,Z 403.508,A -85,B 0,C 180,E1 33624.241,E2 33624.241} C_VEL
LIN {X 0,Y 712.199,Z 403.509,A -85,B 0,C 180,E1 33621.833,E2 33621.833} C_VEL
LIN {X 0,Y 712.278,Z 403.495,A -85,B 0,C 180,E1 33619.037,E2 33619.037} C_VEL
LIN {X 0,Y 712.19,Z 403.509,A -85,B 0,C 180,E1 33616.19,E2 33616.19} C_VEL
LIN {X 0,Y 712.183,Z 403.51,A -85,B 0,C 180,E1 33613.802,E2 33613.802} C_VEL
LIN {X 0,Y 712.247,Z 403.491,A -85,B 0,C 180,E1 33611.072,E2 33611.072} C_VEL
LIN {X 0,Y 712.182,Z 403.505,A -85,B 0,C 180,E1 33608.165,E2 33608.165} C_VEL
LIN {X 0,Y 712.172,Z 403.517,A -85,B 0,C 180,E1 33605.836,E2 33605.836} C_VEL
LIN {X 0,Y 712.186,Z 403.52,A -85,B 0,C 180,E1 33603.488,E2 33603.488} C_VEL
LIN {X 0,Y 712.291,Z 403.883,A -85,B 0,C 180,E1 33603.041,E2 33603.041} C_VEL
LIN {X 0,Y 715.744,Z 413.973,A -85,B 0,C 180,E1 33602.066,E2 33602.066} C_VEL
LIN {X 0,Y 718.323,Z 419.124,A -85,B 0,C 180,E1 33601.853,E2 33601.853} C_VEL
LIN {X 0,Y 719.859,Z 425.585,A -85,B 0,C 180,E1 33601.69,E2 33601.69} C_VEL
LIN {X 0,Y 718.608,Z 676.388,A -85,B 0,C 180,E1 33598.82,E2 33598.82} C_VEL
LIN {X 0,Y 717.999,Z 802.957,A -85,B 0,C 180,E1 33597.377,E2 33597.377} C_VEL
LIN {X 0,Y 717.644,Z 828.386,A -85,B 0,C 180,E1 33596.945,E2 33596.945} C_VEL
LIN {X 0,Y 717.298,Z 850.184,A -85,B 0,C 180,E1 33596.436,E2 33596.436} C_VEL
LIN {X 0,Y 716.884,Z 873.621,A -85,B 0,C 180,E1 33595.752,E2 33595.752} C_VEL
LIN {X 0,Y 716.344,Z 896.305,A -85,B 0,C 180,E1 33594.932,E2 33594.932} C_VEL
LIN {X 0,Y 715.837,Z 919.436,A -85,B 0,C 180,E1 33593.94,E2 33593.94} C_VEL
LIN {X 0,Y 715.251,Z 940.567,A -85,B 0,C 180,E1 33592.87,E2 33592.87} C_VEL
LIN {X 0,Y 714.718,Z 961.85,A -85,B 0,C 180,E1 33591.632,E2 33591.632} C_VEL
LIN {X 0,Y 714.17,Z 981.375,A -85,B 0,C 180,E1 33590.317,E2 33590.317} C_VEL
LIN {X 0,Y 713.707,Z 1000.216,A -85,B 0,C 180,E1 33588.883,E2 33588.883} C_VEL
LIN {X 0,Y 713.293,Z 1016.601,A -85,B 0,C 180,E1 33587.457,E2 33587.457} C_VEL
LIN {X 0,Y 712.929,Z 1033.325,A -85,B 0,C 180,E1 33585.819,E2 33585.819} C_VEL
LIN {X 0,Y 712.61,Z 1047.606,A -85,B 0,C 180,E1 33584.214,E2 33584.214} C_VEL
LIN {X 0,Y 712.402,Z 1061.214,A -85,B 0,C 180,E1 33582.483,E2 33582.483} C_VEL
LIN {X 0,Y 712.205,Z 1073.318,A -85,B 0,C 180,E1 33580.68,E2 33580.68} C_VEL
LIN {X 0,Y 712.07,Z 1084.203,A -85,B 0,C 180,E1 33578.804,E2 33578.804} C_VEL
LIN {X 0,Y 711.973,Z 1092.743,A -85,B 0,C 180,E1 33577.018,E2 33577.018} C_VEL
LIN {X 0,Y 711.936,Z 1099.251,A -85,B 0,C 180,E1 33575.4,E2 33575.4} C_VEL
LIN {X 0,Y 711.9,Z 1105.514,A -85,B 0,C 180,E1 33573.463,E2 33573.463} C_VEL
LIN {X 0,Y 711.916,Z 1109.848,A -85,B 0,C 180,E1 33571.61,E2 33571.61} C_VEL
LIN {X 0,Y 711.905,Z 1112.928,A -85,B 0,C 180,E1 33569.678,E2 33569.678} C_VEL
LIN {X 0,Y 711.901,Z 1114.288,A -85,B 0,C 180,E1 33567.746,E2 33567.746} C_VEL
LIN {X 0,Y 711.902,Z 1114.257,A -85,B 0,C 180,E1 33566.054,E2 33566.054} C_VEL
LIN {X 0,Y 711.915,Z 1112.51,A -85,B 0,C 180,E1 33563.932,E2 33563.932} C_VEL
LIN {X 0,Y 711.919,Z 1109.592,A -85,B 0,C 180,E1 33562.17,E2 33562.17} C_VEL
LIN {X 0,Y 711.915,Z 1104.873,A -85,B 0,C 180,E1 33560.215,E2 33560.215} C_VEL
LIN {X 0,Y 711.932,Z 1098.891,A -85,B 0,C 180,E1 33558.414,E2 33558.414} C_VEL
LIN {X 0,Y 711.986,Z 1092.2,A -85,B 0,C 180,E1 33556.767,E2 33556.767} C_VEL
LIN {X 0,Y 712.074,Z 1082.382,A -85,B 0,C 180,E1 33554.776,E2 33554.776} C_VEL
LIN {X 0,Y 712.212,Z 1072.535,A -85,B 0,C 180,E1 33553.105,E2 33553.105} C_VEL
LIN {X 0,Y 712.422,Z 1059.909,A -85,B 0,C 180,E1 33551.252,E2 33551.252} C_VEL
LIN {X 0,Y 712.627,Z 1046.797,A -85,B 0,C 180,E1 33549.6,E2 33549.6} C_VEL
LIN {X 0,Y 712.958,Z 1031.739,A -85,B 0,C 180,E1 33547.923,E2 33547.923} C_VEL
LIN {X 0,Y 713.319,Z 1015.636,A -85,B 0,C 180,E1 33546.365,E2 33546.365} C_VEL
LIN {X 0,Y 713.751,Z 998.447,A -85,B 0,C 180,E1 33544.883,E2 33544.883} C_VEL
LIN {X 0,Y 714.225,Z 979.723,A -85,B 0,C 180,E1 33543.475,E2 33543.475} C_VEL
LIN {X 0,Y 714.771,Z 958.944,A -85,B 0,C 180,E1 33542.1,E2 33542.1} C_VEL
LIN {X 0,Y 715.315,Z 938.676,A -85,B 0,C 180,E1 33540.938,E2 33540.938} C_VEL
LIN {X 0,Y 715.897,Z 916.02,A -85,B 0,C 180,E1 33539.814,E2 33539.814} C_VEL
LIN {X 0,Y 716.396,Z 894.5,A -85,B 0,C 180,E1 33538.908,E2 33538.908} C_VEL
LIN {X 0,Y 716.942,Z 870.761,A -85,B 0,C 180,E1 33538.067,E2 33538.067} C_VEL
LIN {X 0,Y 717.323,Z 847.855,A -85,B 0,C 180,E1 33537.413,E2 33537.413} C_VEL
LIN {X 0,Y 717.773,Z 823.501,A -85,B 0,C 180,E1 33536.867,E2 33536.867} C_VEL
LIN {X 0,Y 718.011,Z 799.946,A -85,B 0,C 180,E1 33536.493,E2 33536.493} C_VEL
LIN {X 0,Y 719.274,Z 538.908,A -85,B 0,C 180,E1 33533.526,E2 33533.526} C_VEL
LIN {X 0,Y 719.697,Z 424.214,A -85,B 0,C 180,E1 33532.194,E2 33532.194} C_VEL
LIN {X 0,Y 717.684,Z 417.546,A -85,B 0,C 180,E1 33532.003,E2 33532.003} C_VEL
LIN {X 0,Y 715.537,Z 413.496,A -85,B 0,C 180,E1 33531.817,E2 33531.817} C_VEL
LIN {X 0,Y 712.249,Z 403.673,A -85,B 0,C 180,E1 33530.83,E2 33530.83} C_VEL
LIN {X 0,Y 712.175,Z 403.517,A -85,B 0,C 180,E1 33528.204,E2 33528.204} C_VEL
LIN {X 0,Y 712.189,Z 403.515,A -85,B 0,C 180,E1 33525.727,E2 33525.727} C_VEL
LIN {X 0,Y 712.251,Z 403.498,A -85,B 0,C 180,E1 33522.802,E2 33522.802} C_VEL
LIN {X 0,Y 712.189,Z 403.509,A -85,B 0,C 180,E1 33520.123,E2 33520.123} C_VEL
LIN {X 0,Y 712.193,Z 403.51,A -85,B 0,C 180,E1 33517.744,E2 33517.744} C_VEL
LIN {X 0,Y 712.277,Z 403.496,A -85,B 0,C 180,E1 33514.933,E2 33514.933} C_VEL
LIN {X 0,Y 712.204,Z 403.507,A -85,B 0,C 180,E1 33512.052,E2 33512.052} C_VEL
LIN {X 0,Y 712.21,Z 403.492,A -85,B 0,C 180,E1 33509.524,E2 33509.524} C_VEL
LIN {X 0,Y 712.278,Z 403.505,A -85,B 0,C 180,E1 33506.591,E2 33506.591} C_VEL
LIN {X 0,Y 712.211,Z 403.503,A -85,B 0,C 180,E1 33503.761,E2 33503.761} C_VEL
LIN {X 0,Y 712.246,Z 403.511,A -85,B 0,C 180,E1 33501.149,E2 33501.149} C_VEL
LIN {X 0,Y 712.241,Z 403.504,A -85,B 0,C 180,E1 33498.075,E2 33498.075} C_VEL
LIN {X 0,Y 712.226,Z 403.502,A -85,B 0,C 180,E1 33495.387,E2 33495.387} C_VEL
LIN {X 0,Y 712.28,Z 403.5,A -85,B 0,C 180,E1 33492.485,E2 33492.485} C_VEL
LIN {X 0,Y 712.231,Z 403.505,A -85,B 0,C 180,E1 33489.617,E2 33489.617} C_VEL
LIN {X 0,Y 712.283,Z 403.504,A -85,B 0,C 180,E1 33486.772,E2 33486.772} C_VEL
LIN {X 0,Y 712.251,Z 403.502,A -85,B 0,C 180,E1 33483.783,E2 33483.783} C_VEL
LIN {X 0,Y 712.266,Z 403.504,A -85,B 0,C 180,E1 33480.885,E2 33480.885} C_VEL
LIN {X 0,Y 712.261,Z 403.496,A -85,B 0,C 180,E1 33477.747,E2 33477.747} C_VEL
LIN {X 0,Y 712.275,Z 403.509,A -85,B 0,C 180,E1 33474.765,E2 33474.765} C_VEL
LIN {X 0,Y 712.27,Z 403.496,A -85,B 0,C 180,E1 33471.686,E2 33471.686} C_VEL
LIN {X 0,Y 712.276,Z 403.506,A -85,B 0,C 180,E1 33468.666,E2 33468.666} C_VEL
LIN {X 0,Y 712.279,Z 403.499,A -85,B 0,C 180,E1 33465.609,E2 33465.609} C_VEL
LIN {X 0,Y 712.278,Z 403.507,A -85,B 0,C 180,E1 33462.518,E2 33462.518} C_VEL
LIN {X 0,Y 712.275,Z 403.497,A -85,B 0,C 180,E1 33459.445,E2 33459.445} C_VEL
LIN {X 0,Y 712.272,Z 403.51,A -85,B 0,C 180,E1 33456.416,E2 33456.416} C_VEL
LIN {X 0,Y 712.278,Z 403.492,A -85,B 0,C 180,E1 33453.397,E2 33453.397} C_VEL
LIN {X 0,Y 712.268,Z 403.507,A -85,B 0,C 180,E1 33450.339,E2 33450.339} C_VEL
LIN {X 0,Y 712.271,Z 403.499,A -85,B 0,C 180,E1 33447.38,E2 33447.38} C_VEL
LIN {X 0,Y 712.263,Z 403.506,A -85,B 0,C 180,E1 33444.268,E2 33444.268} C_VEL
LIN {X 0,Y 712.266,Z 403.499,A -85,B 0,C 180,E1 33441.309,E2 33441.309} C_VEL
LIN {X 0,Y 712.257,Z 403.504,A -85,B 0,C 180,E1 33438.178,E2 33438.178} C_VEL
LIN {X 0,Y 712.251,Z 403.503,A -85,B 0,C 180,E1 33435.305,E2 33435.305} C_VEL
LIN {X 0,Y 712.269,Z 403.503,A -85,B 0,C 180,E1 33432.255,E2 33432.255} C_VEL
LIN {X 0,Y 712.225,Z 403.504,A -85,B 0,C 180,E1 33429.453,E2 33429.453} C_VEL
LIN {X 0,Y 712.306,Z 403.721,A -85,B 0,C 180,E1 33428.914,E2 33428.914} C_VEL
LIN {X 0,Y 717.903,Z 418.681,A -85,B 0,C 180,E1 33427.449,E2 33427.449} C_VEL
LIN {X 0,Y 717.181,Z 452.736,A -85,B 0,C 180,E1 33425.058,E2 33425.058} C_VEL
LIN {X 0,Y 719.857,Z 464.61,A -85,B 0,C 180,E1 33424.747,E2 33424.747} C_VEL
LIN {X 0,Y 718.606,Z 715.288,A -85,B 0,C 180,E1 33421.878,E2 33421.878} C_VEL
LIN {X 0,Y 718.009,Z 842.945,A -85,B 0,C 180,E1 33420.422,E2 33420.422} C_VEL
LIN {X 0,Y 717.638,Z 868.495,A -85,B 0,C 180,E1 33419.987,E2 33419.987} C_VEL
LIN {X 0,Y 717.29,Z 890.215,A -85,B 0,C 180,E1 33419.48,E2 33419.48} C_VEL
LIN {X 0,Y 716.857,Z 914.562,A -85,B 0,C 180,E1 33418.765,E2 33418.765} C_VEL
LIN {X 0,Y 716.34,Z 936.481,A -85,B 0,C 180,E1 33417.97,E2 33417.97} C_VEL
LIN {X 0,Y 715.831,Z 959.58,A -85,B 0,C 180,E1 33416.978,E2 33416.978} C_VEL
LIN {X 0,Y 715.246,Z 980.753,A -85,B 0,C 180,E1 33415.904,E2 33415.904} C_VEL
LIN {X 0,Y 714.719,Z 1001.753,A -85,B 0,C 180,E1 33414.683,E2 33414.683} C_VEL
LIN {X 0,Y 714.188,Z 1021.128,A -85,B 0,C 180,E1 33413.38,E2 33413.38} C_VEL
LIN {X 0,Y 713.719,Z 1039.823,A -85,B 0,C 180,E1 33411.961,E2 33411.961} C_VEL
LIN {X 0,Y 713.296,Z 1056.461,A -85,B 0,C 180,E1 33410.515,E2 33410.515} C_VEL
LIN {X 0,Y 712.946,Z 1072.964,A -85,B 0,C 180,E1 33408.903,E2 33408.903} C_VEL
LIN {X 0,Y 712.617,Z 1087.221,A -85,B 0,C 180,E1 33407.305,E2 33407.305} C_VEL
LIN {X 0,Y 712.39,Z 1101.059,A -85,B 0,C 180,E1 33405.55,E2 33405.55} C_VEL
LIN {X 0,Y 712.209,Z 1112.796,A -85,B 0,C 180,E1 33403.808,E2 33403.808} C_VEL
LIN {X 0,Y 712.083,Z 1122.948,A -85,B 0,C 180,E1 33402.077,E2 33402.077} C_VEL
LIN {X 0,Y 711.989,Z 1132.538,A -85,B 0,C 180,E1 33400.11,E2 33400.11} C_VEL
LIN {X 0,Y 711.941,Z 1139.119,A -85,B 0,C 180,E1 33398.48,E2 33398.48} C_VEL
LIN {X 0,Y 711.917,Z 1145.451,A -85,B 0,C 180,E1 33396.532,E2 33396.532} C_VEL
LIN {X 0,Y 711.914,Z 1149.814,A -85,B 0,C 180,E1 33394.673,E2 33394.673} C_VEL
LIN {X 0,Y 711.882,Z 1152.685,A -85,B 0,C 180,E1 33392.898,E2 33392.898} C_VEL
LIN {X 0,Y 711.891,Z 1154.262,A -85,B 0,C 180,E1 33390.885,E2 33390.885} C_VEL
LIN {X 0,Y 711.883,Z 1154.306,A -85,B 0,C 180,E1 33389.276,E2 33389.276} C_VEL
LIN {X 0,Y 711.887,Z 1153.017,A -85,B 0,C 180,E1 33387.343,E2 33387.343} C_VEL
LIN {X 0,Y 711.917,Z 1149.972,A -85,B 0,C 180,E1 33385.408,E2 33385.408} C_VEL
LIN {X 0,Y 711.921,Z 1145.864,A -85,B 0,C 180,E1 33383.63,E2 33383.63} C_VEL
LIN {X 0,Y 711.945,Z 1139.423,A -85,B 0,C 180,E1 33381.601,E2 33381.601} C_VEL
LIN {X 0,Y 711.98,Z 1132.892,A -85,B 0,C 180,E1 33379.971,E2 33379.971} C_VEL
LIN {X 0,Y 712.078,Z 1123.866,A -85,B 0,C 180,E1 33378.088,E2 33378.088} C_VEL
LIN {X 0,Y 712.199,Z 1113.317,A -85,B 0,C 180,E1 33376.275,E2 33376.275} C_VEL
LIN {X 0,Y 712.375,Z 1101.641,A -85,B 0,C 180,E1 33374.533,E2 33374.533} C_VEL
LIN {X 0,Y 712.603,Z 1087.928,A -85,B 0,C 180,E1 33372.778,E2 33372.778} C_VEL
LIN {X 0,Y 712.926,Z 1073.741,A -85,B 0,C 180,E1 33371.181,E2 33371.181} C_VEL
LIN {X 0,Y 713.27,Z 1057.39,A -85,B 0,C 180,E1 33369.57,E2 33369.57} C_VEL
LIN {X 0,Y 713.689,Z 1040.776,A -85,B 0,C 180,E1 33368.119,E2 33368.119} C_VEL
